# B&R Automation Studio project PLC code - cp (part 17)

#### MachineModel.st
```iecst
ACTION MachineModel:

	//Assignation of machine model just when unnasigned
	IF gMachine.In.iMachineModelCode=0 THEN
		InputsMachineModel;
	END_IF

	// Code To PLC.
	// From the inputs of the type of machine readed by the inputs to the Parameter of the particular Type of Machine
	MachineModelAssignation;

	//Assignation of the axis
	AxisAssignation;

	// Code To Kernel	(Tranfer the other codes)
	MachineModelCodificationToSw;

END_ACTION

ACTION MachineModelAssignation:

	CASE gMachine.Pt.ConfigNameID OF

		GC_CONFIG_2BK12BAR_ID:
			CASE gMachine.In.iMachineModelCode OF
				51: // P4 Large 1 Block		|| 51-> 0011 0011
					gMachine.Pt.MachineModel:= Type_P4_6B_L;				// 3
				15: // P4 Large 2 Block		|| 15-> 0000 1111
					gMachine.Pt.MachineModel:=Type_P4_12B_L;				// 4
				48: // P4 Short 1 Block		|| 48-> 0011 0000
					gMachine.Pt.MachineModel:=Type_P4_6B;					// 1
				11: //S1400 Without Vacuum	|| 11-> 0000 1011
					gMachine.Pt.MachineModel:=Type_P4_CBK;					// 14
				12: // P4 Short 2 Block		|| 12-> 0000 1100
					gMachine.Pt.MachineModel:=Type_P4_12B;					// 2
				52: // P4 Long 1 Block Cubik|| 11-> 0011 0100
					gMachine.Pt.MachineModel:= Type_P4_CBK;				// 12 -->P4 1 Block normal with vacuum and cubik functions
				ELSE
					gMachine.Pt.MachineModel:=NoType;

			END_CASE

		GC_CONFIG_1BK2BAR_ID:
			CASE gMachine.In.iMachineModelCode OF
				3: // EBRO 1 Block			|| 3->  0000 0011
					gMachine.Pt.MachineModel:=Type_SHLD;					// 5
				ELSE
					gMachine.Pt.MachineModel:=NoType;

			END_CASE

		GC_CONFIG_BM_1BK8BAR_ID:
			CASE gMachine.In.iMachineModelCode OF
				5: //P5 Oil					|| 5->	0000 0101
					gMachine.Pt.MachineModel:=Type_P5_OIL;
				6: //P5 Water				|| 6->	0000 0110
					gMachine.Pt.MachineModel:=Type_P5_WTR;
				13: //S1400 Without Vacuum	|| 13-> 0000 1101
					gMachine.Pt.MachineModel:=Type_S1400;
				14: //S1400 With Vacuum	PWRLNK	|| 14->	0000 1110
					gMachine.Pt.MachineModel:=Type_S1400_VAC_PWRLNK;
				15: //S1400 With Vacuum	CAN		|| 14->	0000 1111
					gMachine.Pt.MachineModel:=Type_S1400_VAC_CAN;

				ELSE
					gMachine.Pt.MachineModel:=NoType;

			END_CASE

		GC_CONFIG_1BK8BAR_NOZ2_ID:
			CASE gMachine.In.iMachineModelCode OF
				40:
					gMachine.Pt.MachineModel:=Type_NOZ_2_UV;				// 15
				41:
					gMachine.Pt.MachineModel:=Type_NOZ_2_UV_White;

				ELSE
					gMachine.Pt.MachineModel:=NoType;

			END_CASE

		GC_CONFIG_1BK8BAR_NOZ2_AQ_ID:
			CASE gMachine.In.iMachineModelCode OF
				39:
					gMachine.Pt.MachineModel:=Type_NOZ_2_AQ;

				ELSE
					gMachine.Pt.MachineModel:=NoType;

			END_CASE

		GC_CONFIG_1BK7BAR_CUBE_ID:
			CASE gMachine.In.iMachineModelCode OF
				01:
					gMachine.Pt.MachineModel:=Type_CUBE_INSPECTION;
				02:
					gMachine.Pt.MachineModel := Type_CUBE_GULLIVER_INSPECTION;
				04:
					gMachine.Pt.MachineModel:=Type_CUBE;
				08:
					gMachine.Pt.MachineModel := Type_CUBE_GULLIVER;
				ELSE
					gMachine.Pt.MachineModel:=NoType;

			END_CASE

		GC_CONFIG_1BK10BAR_MECANO_ID:
			CASE gMachine.In.iMachineModelCode OF
				60:
					gMachine.Pt.MachineModel:=Type_MECANO_UV_WHITE;
				61:
					gMachine.Pt.MachineModel:=Type_MECANO_UV_OPV;
				62:
					gMachine.Pt.MachineModel:=Type_MECANO_UV_WHITE_OPV;

				ELSE
					gMachine.Pt.MachineModel:=NoType;

			END_CASE

		GC_CONFIG_SIMTEST_ID:
			CASE gMachine.In.iMachineModelCode OF
				51: // P4 Large 1 Block		|| 51-> 0011 0011
					gMachine.Pt.MachineModel:= Type_P4_6B_L;				// 3
				15: // P4 Large 2 Block		|| 15-> 0000 1111
					gMachine.Pt.MachineModel:=Type_P4_12B_L;				// 4
				48: // P4 Short 1 Block		|| 48-> 0011 0000
					gMachine.Pt.MachineModel:=Type_P4_6B;					// 1
				12: // P4 Short 2 Block		|| 12-> 0000 0011
					gMachine.Pt.MachineModel:=Type_P4_12B;					// 2
				3: // EBRO 1 Block			|| 3->  0000 0011
					gMachine.Pt.MachineModel:=Type_SHLD;					// 5
				13: //S1400 Without Vacuum	|| 13-> 0000 1011
					gMachine.Pt.MachineModel:=Type_S1400;					// 9
				14: //S1400 With Vacuum	PWLNK
					gMachine.Pt.MachineModel:=Type_S1400_VAC_PWRLNK;
				1015: //S1400 With Vacuum CAN
					gMachine.Pt.MachineModel:=Type_S1400_VAC_PWRLNK;
				52: // P4 Long 1 Block Cubik|| 11-> 0011 0100
					gMachine.Pt.MachineModel:= Type_P4_CBK;				// 12 -->P4 1 Block normal with vacuum and cubik functions
				5: //P5 Oil					|| 5->	0000 0101
					gMachine.Pt.MachineModel:=Type_P5_OIL;					// 12
				6: //P5 Water				|| 6->	0000 0110
					gMachine.Pt.MachineModel:=Type_P5_WTR;					// 13
				11: //S1400 Without Vacuum	|| 11-> 0000 1011
					gMachine.Pt.MachineModel:=Type_P4_CBK;					// 14
				39:
					gMachine.Pt.MachineModel:=Type_NOZ_2_AQ;					// 11
				40:
					gMachine.Pt.MachineModel:=Type_NOZ_2_UV;				// 15
				41:
					gMachine.Pt.MachineModel:=Type_NOZ_2_UV_White;
				60:
					gMachine.Pt.MachineModel:=Type_MECANO_UV_WHITE;
				61:
					gMachine.Pt.MachineModel:=Type_MECANO_UV_OPV;
				62:
					gMachine.Pt.MachineModel:=Type_MECANO_UV_WHITE_OPV;

				10001:
					gMachine.Pt.MachineModel := Type_CUBE;
				10002:
					gMachine.Pt.MachineModel := Type_CUBE_GULLIVER;
				10003:
					gMachine.Pt.MachineModel := Type_CUBE_INSPECTION;
				10004:
					gMachine.Pt.MachineModel := Type_CUBE_GULLIVER_INSPECTION;

				ELSE
					gMachine.Pt.MachineModel:=NoType;

			END_CASE
			xChangedSimMachine := simMachine_copy <> gSimMachine.Parameters.MachineType;
			simMachine_copy := gSimMachine.Parameters.MachineType;

		ELSE
			gMachine.Pt.MachineModel:=NoType;

	END_CASE

END_ACTION

ACTION AxisAssignation:

	IF gMachine.Pt.ConfigNameID = GC_CONFIG_SIMTEST_ID THEN
		Axis_Simulation;
		RETURN;
	END_IF

    //Name of the Axis as defined in Hardware
	CASE gMachine.Pt.MachineModel OF

		Type_P4_6B,
		Type_P4_6B_L,
		Type_P4_12B,
		Type_P4_12B_L:
			Axis_P4;

		Type_SHLD,
		Type_SHLD_L:
			Axis_Shield;

		Type_S1400,
		Type_S1400_VAC_PWRLNK,
		Type_S1400_VAC_CAN:
			Axis_S1400;

		Type_P5_OIL,
		Type_P5_WTR:
			Axis_P5;

		Type_NOZ_2_AQ:
			Axis_Nozomi2_AQ;

		Type_NOZ_2_UV,
		Type_NOZ_2_UV_White:
			Axis_Nozomi2;

		Type_CUBE,
		Type_CUBE_INSPECTION,
		Type_CUBE_GULLIVER,
		Type_CUBE_GULLIVER_INSPECTION:
			Axis_Cube;

		Type_MECANO_UV_WHITE,
		Type_MECANO_UV_OPV,
		Type_MECANO_UV_WHITE_OPV:
			Axis_Mecano;

		ELSE
			//No machine assigned
			RETURN;

	END_CASE

END_ACTION

ACTION Axis_Simulation:

	gAxis[1].Parameter.Init.AxisObjectName			:=	'gAxis01';	//Instance_Belt
	gAxis[2].Parameter.Init.AxisObjectName			:=	'gAxis21';	//Instance_BK1
	gAxis[3].Parameter.Init.AxisObjectName			:=	'gAxis121';	//Instance_BK2
	gAxis[4].Parameter.Init.AxisObjectName			:=	'gAxisStp01';	//Instance_Front3L
	gAxis[5].Parameter.Init.AxisObjectName			:=	'gAxisStp02';	//Instance_Back3L
	gAxis[6].Parameter.Init.AxisObjectName			:=	'gAxis41';	//Instance_NonCrash1

	// Assignation of Master axis
	gAxis[5].Parameter.Init.MasterGearObjectName	:=	'gAxisStp01';	//Instance_Front3L

	LoadDefaultServoConfig(ADR(gAxis[1]));
	LoadDefaultServoConfig(ADR(gAxis[2]));
	LoadDefaultServoConfig(ADR(gAxis[3]));
	LoadDefaultStepperConfig(ADR(gAxis[4])); //These are steppers and do not have torque
	LoadDefaultStepperConfig(ADR(gAxis[5])); //These are steppers and do not have torque
	LoadDefaultServoConfig(ADR(gAxis[6]));

	//Assign comms type of inverters depending on the machine type
	CASE gMachine.Pt.MachineModel OF
		Type_S1400_VAC_PWRLNK:
			gAxisInverter[1].Parameters.CommsType := COMMS_POWERLINK;
			gAxisInverter[2].Parameters.CommsType := COMMS_POWERLINK;
			gAxisInverter[3].Parameters.CommsType := COMMS_POWERLINK;
			gAxisInverter[4].Parameters.CommsType := COMMS_POWERLINK;

		Type_NOZ_2_AQ:
			IF X20IF1072_SS3.ModuleOk THEN
				gAxisInverter[1].Parameters.CommsType := COMMS_CANOPEN;
				gAxisInverter[2].Parameters.CommsType := COMMS_CANOPEN;
				gAxisInverter[3].Parameters.CommsType := COMMS_CANOPEN;
				gAxisInverter[4].Parameters.CommsType := COMMS_CANOPEN;
			ELSE
				gAxisInverter[1].Parameters.CommsType := COMMS_POWERLINK;
				gAxisInverter[2].Parameters.CommsType := COMMS_POWERLINK;
				gAxisInverter[3].Parameters.CommsType := COMMS_POWERLINK;
				gAxisInverter[4].Parameters.CommsType := COMMS_POWERLINK;
			END_IF

		Type_NOZ_2_UV,
		Type_NOZ_2_UV_White:
			IF X20IF1072_SS1.ModuleOk THEN
				gAxisInverter[1].Parameters.CommsType := COMMS_CANOPEN;
				gAxisInverter[2].Parameters.CommsType := COMMS_CANOPEN;
				gAxisInverter[3].Parameters.CommsType := COMMS_CANOPEN;
				gAxisInverter[4].Parameters.CommsType := COMMS_CANOPEN;
			ELSE
				gAxisInverter[1].Parameters.CommsType := COMMS_POWERLINK;
				gAxisInverter[2].Parameters.CommsType := COMMS_POWERLINK;
				gAxisInverter[3].Parameters.CommsType := COMMS_POWERLINK;
				gAxisInverter[4].Parameters.CommsType := COMMS_POWERLINK;
			END_IF

		Type_CUBE,
		Type_CUBE_INSPECTION,
		Type_CUBE_GULLIVER,
		Type_CUBE_GULLIVER_INSPECTION:
			gAxisInverter[1].Parameters.CommsType := COMMS_POWERLINK;
			gAxisInverter[2].Parameters.CommsType := COMMS_POWERLINK;
			gAxisInverter[3].Parameters.CommsType := COMMS_POWERLINK;

		Type_MECANO_UV_WHITE,
		Type_MECANO_UV_OPV,
		Type_MECANO_UV_WHITE_OPV:
			gAxisInverter[1].Parameters.CommsType := COMMS_POWERLINK;
			gAxisInverter[2].Parameters.CommsType := COMMS_POWERLINK;
			gAxisInverter[3].Parameters.CommsType := COMMS_POWERLINK;
			gAxisInverter[4].Parameters.CommsType := COMMS_POWERLINK;

	END_CASE
	gAxisInverter[1].Parameters.Hardware.CpuFamily := gMachine.St.HwData.Family;
	gAxisInverter[2].Parameters.Hardware.CpuFamily := gMachine.St.HwData.Family;
	gAxisInverter[3].Parameters.Hardware.CpuFamily := gMachine.St.HwData.Family;
	gAxisInverter[4].Parameters.Hardware.CpuFamily := gMachine.St.HwData.Family;

	//This is the physical node of each Icla
	gIcla[1].Parameter.Node:=5;
	gIcla[1].Parameter.Network := 'IF7';
	gIcla[2].Parameter.Node:=7;
	gIcla[2].Parameter.Network := 'IF7';
	gIcla[3].Parameter.Node:=50; //Same node number than in Nozomi C18000
	gIcla[3].Parameter.Network := 'IF7';

END_ACTION

ACTION Axis_P4:

	gAxis[1].Parameter.Init.AxisObjectName			:=	'gAxis01';	//Instance_Belt
	gAxis[2].Parameter.Init.AxisObjectName			:=	'gAxis21';	//Instance_BK1
	gAxis[3].Parameter.Init.AxisObjectName			:=	'gAxis121';	//Instance_BK2
	gAxis[4].Parameter.Init.AxisObjectName			:=	'gAxisStp01';	//Instance_Front3L
	gAxis[5].Parameter.Init.AxisObjectName			:=	'gAxisStp02';	//Instance_Back3L

	// Assignation of Master axis
	gAxis[5].Parameter.Init.MasterGearObjectName	:=	'gAxisStp01';	//Instance_Front3L

	LoadDefaultServoConfig(ADR(gAxis[1]));
	LoadDefaultServoConfig(ADR(gAxis[2]));
	LoadDefaultServoConfig(ADR(gAxis[3]));
	LoadDefaultStepperConfig(ADR(gAxis[4])); //These are steppers and do not have torque
	LoadDefaultStepperConfig(ADR(gAxis[5])); //These are steppers and do not have torque

	//This is the physical node of each Icla
	gIcla[1].Parameter.Node:=5;
	gIcla[1].Parameter.Network := 'IF7';
	gIcla[1].Parameter.xAutoresetComms := TRUE;
	gIcla[2].Parameter.Node:=7;
	gIcla[2].Parameter.Network := 'IF7';
	gIcla[2].Parameter.xAutoresetComms := TRUE;

END_ACTION

ACTION Axis_Shield:

	gAxis[1].Parameter.Init.AxisObjectName			:=	'gAxis01';	//Instance_Belt
	gAxis[2].Parameter.Init.AxisObjectName			:=	'gAxis21';	//Instance_BK1
	gAxis[3].Parameter.Init.AxisObjectName			:=	'gAxisStp01';	//Instance_Front3L
	gAxis[4].Parameter.Init.AxisObjectName			:=	'gAxisStp02';	//Instance_Back3L

	// Assignation of Master axis
	gAxis[4].Parameter.Init.MasterGearObjectName	:=	'gAxisStp01';	//Instance_Front3L

	LoadDefaultServoConfig(ADR(gAxis[1]));
	LoadDefaultServoConfig(ADR(gAxis[2]));
	LoadDefaultStepperConfig(ADR(gAxis[3])); //These are steppers and do not have torque
	LoadDefaultStepperConfig(ADR(gAxis[4])); //These are steppers and do not have torque

	//This is the physical node of each Icla
	gIcla[1].Parameter.Node:=5;
	gIcla[1].Parameter.Network := 'IF7';
	gIcla[1].Parameter.xAutoresetComms := TRUE;

END_ACTION

ACTION Axis_S1400:

	gAxis[1].Parameter.Init.AxisObjectName			:=	'gAxis01';	//Instance_Belt
	gAxis[2].Parameter.Init.AxisObjectName			:=	'gAxis21';	//Instance_BK1
	gAxis[3].Parameter.Init.AxisObjectName			:=	'gAxisStp01';	//Instance_Front3L
	gAxis[4].Parameter.Init.AxisObjectName			:=	'gAxisStp02';	//Instance_Back3L
	gAxis[5].Parameter.Init.AxisObjectName			:=	'gAxis41';	//Instance_NonCrash1

	// Assignation of Master axis
	gAxis[4].Parameter.Init.MasterGearObjectName	:=	'gAxisStp01';	//Instance_Front3L

	CASE gMachine.Pt.MachineModel OF
		Type_S1400_VAC_PWRLNK:
			gAxisInverter[1].Parameters.Hardware.PowerLinkInterface := 'IF3';
			gAxisInverter[1].Parameters.Hardware.Node := 81;
			gAxisInverter[1].Parameters.AccelerationTime := 1;
			gAxisInverter[1].Parameters.DecelerationTime := 1;
			gAxisInverter[1].Parameters.CommsType := COMMS_POWERLINK;
			gAxisInverter[2].Parameters.Hardware.PowerLinkInterface := 'IF3';
			gAxisInverter[2].Parameters.Hardware.Node := 82;
			gAxisInverter[2].Parameters.AccelerationTime := 1;
			gAxisInverter[2].Parameters.DecelerationTime := 1;
			gAxisInverter[2].Parameters.CommsType := COMMS_POWERLINK;
			gAxisInverter[3].Parameters.Hardware.PowerLinkInterface := 'IF3';
			gAxisInverter[3].Parameters.Hardware.Node := 83;
			gAxisInverter[3].Parameters.AccelerationTime := 1;
			gAxisInverter[3].Parameters.DecelerationTime := 1;
			gAxisInverter[3].Parameters.CommsType := COMMS_POWERLINK;
			gAxisInverter[4].Parameters.Hardware.PowerLinkInterface := 'IF3';
			gAxisInverter[4].Parameters.Hardware.Node := 84;
			gAxisInverter[4].Parameters.AccelerationTime := 1;
			gAxisInverter[4].Parameters.DecelerationTime := 1;
			gAxisInverter[4].Parameters.CommsType := COMMS_POWERLINK;

		Type_S1400_VAC_CAN:
			gAxisInverter[1].Parameters.CommsType := COMMS_CANOPEN;
			gAxisInverter[2].Parameters.CommsType := COMMS_CANOPEN;
			gAxisInverter[3].Parameters.CommsType := COMMS_CANOPEN;
			gAxisInverter[4].Parameters.CommsType := COMMS_CANOPEN;

	END_CASE

	gAxisInverter[1].Parameters.Hardware.CpuFamily := gMachine.St.HwData.Family;
	gAxisInverter[2].Parameters.Hardware.CpuFamily := gMachine.St.HwData.Family;
	gAxisInverter[3].Parameters.Hardware.CpuFamily := gMachine.St.HwData.Family;
	gAxisInverter[4].Parameters.Hardware.CpuFamily := gMachine.St.HwData.Family;

	LoadDefaultServoConfig(ADR(gAxis[1]));
	LoadDefaultServoConfig(ADR(gAxis[2]));
	LoadDefaultStepperConfig(ADR(gAxis[3])); //These are steppers and do not have torque
	LoadDefaultStepperConfig(ADR(gAxis[4])); //These are steppers and do not have torque
	LoadDefaultServoConfig(ADR(gAxis[5]));

	//This is the physical node of each Icla
	gIcla[1].Parameter.Node:=5;
	gIcla[1].Parameter.Network := 'IF7';
	gIcla[1].Parameter.xAutoresetComms := TRUE;

END_ACTION

ACTION Axis_P5:

	gAxis[1].Parameter.Init.AxisObjectName			:=	'gAxis02';	//Instance_Belt
	gAxis[2].Parameter.Init.AxisObjectName			:=	'gAxis21';	//Instance_BK1
	gAxis[3].Parameter.Init.AxisObjectName			:=	'gAxisStp01';	//Instance_Front3L
	gAxis[4].Parameter.Init.AxisObjectName			:=	'gAxisStp02';	//Instance_Back3L

	// Assignation of Master axis
	gAxis[4].Parameter.Init.MasterGearObjectName	:=	'gAxisStp01';	//Instance_Front3L

	LoadDefaultServoConfig(ADR(gAxis[1]));
	LoadDefaultServoConfig(ADR(gAxis[2]));
	LoadDefaultStepperConfig(ADR(gAxis[3])); //These are steppers and do not have torque
	LoadDefaultStepperConfig(ADR(gAxis[4])); //These are steppers and do not have torque

	//This is the physical node of each Icla
	gIcla[1].Parameter.Node:=5;
	gIcla[1].Parameter.Network := 'IF7';
	gIcla[1].Parameter.xAutoresetComms := TRUE;

END_ACTION

ACTION Axis_Nozomi2:

	gAxis[1].Parameter.Init.AxisObjectName			:=	'gAxis01';	//Instance_Belt
	gAxis[2].Parameter.Init.AxisObjectName			:=	'gAxis21';	//Instance_BK1

	LoadDefaultServoConfig(ADR(gAxis[1]));
	LoadDefaultServoConfig(ADR(gAxis[2]));

	CASE gMachine.Pt.MachineModel OF
		Type_NOZ_2_UV,
		Type_NOZ_2_UV_White:

			IF X20IF1072_SS1.ModuleOk THEN
				gAxisInverter[1].Parameters.CommsType := COMMS_CANOPEN;
				gAxisInverter[1].Parameters.Hardware.Node := 81;
				gAxisInverter[1].Parameters.Hardware.PowerLinkInterface := 'IF1';
				gAxisInverter[2].Parameters.CommsType := COMMS_CANOPEN;
				gAxisInverter[2].Parameters.Hardware.Node := 82;
				gAxisInverter[2].Parameters.Hardware.PowerLinkInterface := 'IF1';
				gAxisInverter[3].Parameters.CommsType := COMMS_CANOPEN;
				gAxisInverter[3].Parameters.Hardware.Node := 83;
				gAxisInverter[3].Parameters.Hardware.PowerLinkInterface := 'IF1';
				gAxisInverter[4].Parameters.CommsType := COMMS_CANOPEN;
				gAxisInverter[4].Parameters.Hardware.Node := 84;
				gAxisInverter[4].Parameters.Hardware.PowerLinkInterface := 'IF1';
			ELSE
				gAxisInverter[1].Parameters.Hardware.PowerLinkInterface := 'IF3';
				gAxisInverter[1].Parameters.Hardware.Node := 81;
				gAxisInverter[1].Parameters.AccelerationTime := 3;
				gAxisInverter[1].Parameters.DecelerationTime := 1;
				gAxisInverter[1].Parameters.CommsType := COMMS_POWERLINK;
				gAxisInverter[2].Parameters.Hardware.PowerLinkInterface := 'IF3';
				gAxisInverter[2].Parameters.Hardware.Node := 82;
				gAxisInverter[2].Parameters.AccelerationTime := gAxisInverter[1].Parameters.AccelerationTime;
				gAxisInverter[2].Parameters.DecelerationTime := gAxisInverter[1].Parameters.DecelerationTime;
				gAxisInverter[2].Parameters.CommsType := COMMS_POWERLINK;
				gAxisInverter[3].Parameters.Hardware.PowerLinkInterface := 'IF3';
				gAxisInverter[3].Parameters.Hardware.Node := 83;
				gAxisInverter[3].Parameters.AccelerationTime := gAxisInverter[1].Parameters.AccelerationTime;
				gAxisInverter[3].Parameters.DecelerationTime := gAxisInverter[1].Parameters.DecelerationTime;
				gAxisInverter[3].Parameters.CommsType := COMMS_POWERLINK;
				gAxisInverter[4].Parameters.Hardware.PowerLinkInterface := 'IF3';
				gAxisInverter[4].Parameters.Hardware.Node := 84;
				gAxisInverter[4].Parameters.AccelerationTime := gAxisInverter[1].Parameters.AccelerationTime;
				gAxisInverter[4].Parameters.DecelerationTime := gAxisInverter[1].Parameters.DecelerationTime;
				gAxisInverter[4].Parameters.CommsType := COMMS_POWERLINK;
			END_IF

	END_CASE

	gAxisInverter[1].Parameters.Hardware.CpuFamily := gMachine.St.HwData.Family;
	gAxisInverter[2].Parameters.Hardware.CpuFamily := gMachine.St.HwData.Family;
	gAxisInverter[3].Parameters.Hardware.CpuFamily := gMachine.St.HwData.Family;
	gAxisInverter[4].Parameters.Hardware.CpuFamily := gMachine.St.HwData.Family;

	//This is the physical node of each Icla
	gIcla[1].Parameter.Node:=5;
	gIcla[1].Parameter.Network := 'IF7';
	gIcla[1].Parameter.xAutoresetComms := TRUE;
	gIcla[2].Parameter.Node:=2; //50; [RGP] We had to change number node to match the node order that AS was expecting. Escalated to JNovella. No reason explained.
	gIcla[2].Parameter.Network := 'IF7';
	gIcla[2].Parameter.xAutoresetComms := TRUE;
	gIcla[3].Parameter.Node:=6;
	gIcla[3].Parameter.Network := 'IF7';
	gIcla[3].Parameter.xAutoresetComms := TRUE;
	gIcla[4].Parameter.Node:=7;
	gIcla[4].Parameter.Network := 'IF7';
	gIcla[4].Parameter.xAutoresetComms := TRUE;
	gIcla[5].Parameter.Node:=8;
	gIcla[5].Parameter.Network := 'IF7';
	gIcla[5].Parameter.xAutoresetComms := TRUE;
	gIcla[6].Parameter.Node:=9;
	gIcla[6].Parameter.Network := 'IF7';
	gIcla[6].Parameter.xAutoresetComms := TRUE;

END_ACTION

ACTION Axis_Nozomi2_AQ:

	gAxis[1].Parameter.Init.AxisObjectName			:=	'gAxis01';	//Instance_Belt
	gAxis[2].Parameter.Init.AxisObjectName			:=	'gAxis21';	//Instance_BK1

	LoadDefaultServoConfig(ADR(gAxis[1]));
	LoadDefaultServoConfig(ADR(gAxis[2]));

	CASE gMachine.Pt.MachineModel OF
		Type_NOZ_2_AQ:

			IF X20IF1072_SS3.ModuleOk THEN
				gAxisInverter[1].Parameters.CommsType := COMMS_CANOPEN;
				gAxisInverter[1].Parameters.Hardware.Node := 81;
				gAxisInverter[1].Parameters.Hardware.PowerLinkInterface := 'SS3.IF1';
				gAxisInverter[2].Parameters.CommsType := COMMS_CANOPEN;
				gAxisInverter[2].Parameters.Hardware.Node := 82;
				gAxisInverter[2].Parameters.Hardware.PowerLinkInterface := 'SS3.IF1';
				gAxisInverter[3].Parameters.CommsType := COMMS_CANOPEN;
				gAxisInverter[3].Parameters.Hardware.Node := 83;
				gAxisInverter[3].Parameters.Hardware.PowerLinkInterface := 'SS3.IF1';
				gAxisInverter[4].Parameters.CommsType := COMMS_CANOPEN;
				gAxisInverter[4].Parameters.Hardware.Node := 84;
				gAxisInverter[4].Parameters.Hardware.PowerLinkInterface := 'SS3.IF1';
			ELSE
				gAxisInverter[1].Parameters.Hardware.PowerLinkInterface := 'IF3';
				gAxisInverter[1].Parameters.Hardware.Node := 81;
				gAxisInverter[1].Parameters.AccelerationTime := 3;
				gAxisInverter[1].Parameters.DecelerationTime := 1;
				gAxisInverter[1].Parameters.CommsType := COMMS_POWERLINK;
				gAxisInverter[2].Parameters.Hardware.PowerLinkInterface := 'IF3';
				gAxisInverter[2].Parameters.Hardware.Node := 82;
				gAxisInverter[2].Parameters.AccelerationTime := gAxisInverter[1].Parameters.AccelerationTime;
				gAxisInverter[2].Parameters.DecelerationTime := gAxisInverter[1].Parameters.DecelerationTime;
				gAxisInverter[2].Parameters.CommsType := COMMS_POWERLINK;
				gAxisInverter[3].Parameters.Hardware.PowerLinkInterface := 'IF3';
				gAxisInverter[3].Parameters.Hardware.Node := 83;
				gAxisInverter[3].Parameters.AccelerationTime := gAxisInverter[1].Parameters.AccelerationTime;
				gAxisInverter[3].Parameters.DecelerationTime := gAxisInverter[1].Parameters.DecelerationTime;
				gAxisInverter[3].Parameters.CommsType := COMMS_POWERLINK;
				gAxisInverter[4].Parameters.Hardware.PowerLinkInterface := 'IF3';
				gAxisInverter[4].Parameters.Hardware.Node := 84;
				gAxisInverter[4].Parameters.AccelerationTime := gAxisInverter[1].Parameters.AccelerationTime;
				gAxisInverter[4].Parameters.DecelerationTime := gAxisInverter[1].Parameters.DecelerationTime;
				gAxisInverter[4].Parameters.CommsType := COMMS_POWERLINK;
			END_IF

	END_CASE

	gAxisInverter[1].Parameters.Hardware.CpuFamily := gMachine.St.HwData.Family;
	gAxisInverter[2].Parameters.Hardware.CpuFamily := gMachine.St.HwData.Family;
	gAxisInverter[3].Parameters.Hardware.CpuFamily := gMachine.St.HwData.Family;
	gAxisInverter[4].Parameters.Hardware.CpuFamily := gMachine.St.HwData.Family;

	//This is the physical node of each Icla
	gIcla[1].Parameter.Node:=5;
	gIcla[1].Parameter.Network := 'SS2.IF1';
	gIcla[1].Parameter.xAutoresetComms := TRUE;
	gIcla[2].Parameter.Node:=2; //50; [RGP] We had to change number node to match the node order that AS was expecting. Escalated to JNovella. No reason explained.
	gIcla[2].Parameter.Network := 'SS2.IF1';
	gIcla[2].Parameter.xAutoresetComms := TRUE;
	gIcla[3].Parameter.Node:=6;
	gIcla[3].Parameter.Network := 'SS2.IF1';
	gIcla[3].Parameter.xAutoresetComms := TRUE;
	gIcla[4].Parameter.Node:=7;
	gIcla[4].Parameter.Network := 'SS2.IF1';
	gIcla[4].Parameter.xAutoresetComms := TRUE;
	gIcla[5].Parameter.Node:=8;
	gIcla[5].Parameter.Network := 'SS2.IF1';
	gIcla[5].Parameter.xAutoresetComms := TRUE;
	gIcla[6].Parameter.Node:=9;
	gIcla[6].Parameter.Network := 'SS2.IF1';
	gIcla[6].Parameter.xAutoresetComms := TRUE;

END_ACTION

ACTION Axis_Cube:

	gAxis[1].Parameter.Init.AxisObjectName			:=	'gAxis01';	//Instance_Belt
	gAxis[2].Parameter.Init.AxisObjectName			:=	'gAxis21';	//Instance_BK1

	LoadDefaultServoConfig(ADR(gAxis[1]));
	LoadDefaultServoConfig(ADR(gAxis[2]));

	CASE gMachine.Pt.MachineModel OF
		Type_CUBE,
		Type_CUBE_INSPECTION,
		Type_CUBE_GULLIVER,
		Type_CUBE_GULLIVER_INSPECTION:

			gAxisInverter[1].Parameters.Hardware.PowerLinkInterface := 'IF3';
			gAxisInverter[1].Parameters.Hardware.Node := 81;
			gAxisInverter[1].Parameters.AccelerationTime := 0;
			gAxisInverter[1].Parameters.DecelerationTime := 0;
			gAxisInverter[1].Parameters.CommsType := COMMS_POWERLINK;
			gAxisInverter[1].Parameters.Type := INV_ABB;
			gAxisInverter[1].Parameters.ControlMode := 0;
			gAxisInverter[2].Parameters.Hardware.PowerLinkInterface := 'IF3';
			gAxisInverter[2].Parameters.Hardware.Node := 82;
			gAxisInverter[2].Parameters.AccelerationTime := 0;
			gAxisInverter[2].Parameters.DecelerationTime := 0;
			gAxisInverter[2].Parameters.CommsType := COMMS_POWERLINK;
			gAxisInverter[2].Parameters.Type := INV_ABB;
			gAxisInverter[2].Parameters.ControlMode := 0;

			gAxisInverter[3].Parameters.Hardware.PowerLinkInterface := 'IF3';
			gAxisInverter[3].Parameters.Hardware.Node := 91;
			gAxisInverter[3].Parameters.AccelerationTime := 0;
			gAxisInverter[3].Parameters.DecelerationTime := 0;
			gAxisInverter[3].Parameters.CommsType := COMMS_POWERLINK;
			gAxisInverter[3].Parameters.Type := INV_ABB;
			gAxisInverter[3].Parameters.ControlMode := 0;

	END_CASE

	gAxisInverter[1].Parameters.Hardware.CpuFamily := gMachine.St.HwData.Family;
	gAxisInverter[2].Parameters.Hardware.CpuFamily := gMachine.St.HwData.Family;
	gAxisInverter[3].Parameters.Hardware.CpuFamily := gMachine.St.HwData.Family;

	//This is the physical node of each Icla
	gIcla[1].Parameter.Node:=5;
	gIcla[1].Parameter.Network := 'SS2.IF1';
	gIcla[1].Parameter.xAutoresetComms := TRUE;

END_ACTION

ACTION Axis_Mecano:

	gAxis[1].Parameter.Init.AxisObjectName			:=	'gAxis01';	//Instance_Belt
	gAxis[2].Parameter.Init.AxisObjectName			:=	'gAxis21';	//Instance_BK1

	LoadDefaultServoConfig(ADR(gAxis[1]));
	LoadDefaultServoConfig(ADR(gAxis[2]));

	gAxisInverter[1].Parameters.Hardware.PowerLinkInterface := 'IF3';
	gAxisInverter[1].Parameters.Hardware.Node := 81;
	gAxisInverter[1].Parameters.AccelerationTime := 0;
	gAxisInverter[1].Parameters.DecelerationTime := 0;
	gAxisInverter[1].Parameters.CommsType := COMMS_POWERLINK;
	gAxisInverter[1].Parameters.Type := INV_ABB;
	gAxisInverter[1].Parameters.ControlMode := 0;
	gAxisInverter[2].Parameters.Hardware.PowerLinkInterface := 'IF3';
	gAxisInverter[2].Parameters.Hardware.Node := 82;
	gAxisInverter[2].Parameters.AccelerationTime := 0;
	gAxisInverter[2].Parameters.DecelerationTime := 0;
	gAxisInverter[2].Parameters.CommsType := COMMS_POWERLINK;
	gAxisInverter[2].Parameters.Type := INV_ABB;
	gAxisInverter[2].Parameters.ControlMode := 0;
	gAxisInverter[3].Parameters.Hardware.PowerLinkInterface := 'IF3';
	gAxisInverter[3].Parameters.Hardware.Node := 83;
	gAxisInverter[3].Parameters.AccelerationTime := 0;
	gAxisInverter[3].Parameters.DecelerationTime := 0;
	gAxisInverter[3].Parameters.CommsType := COMMS_POWERLINK;
	gAxisInverter[3].Parameters.Type := INV_ABB;
	gAxisInverter[3].Parameters.ControlMode := 0;
	gAxisInverter[4].Parameters.Hardware.PowerLinkInterface := 'IF3';
	gAxisInverter[4].Parameters.Hardware.Node := 84;
	gAxisInverter[4].Parameters.AccelerationTime := 0;
	gAxisInverter[4].Parameters.DecelerationTime := 0;
	gAxisInverter[4].Parameters.CommsType := COMMS_POWERLINK;
	gAxisInverter[4].Parameters.Type := INV_ABB;
	gAxisInverter[4].Parameters.ControlMode := 0;

	gAxisInverter[1].Parameters.Hardware.CpuFamily := gMachine.St.HwData.Family;
	gAxisInverter[2].Parameters.Hardware.CpuFamily := gMachine.St.HwData.Family;
	gAxisInverter[3].Parameters.Hardware.CpuFamily := gMachine.St.HwData.Family;
	gAxisInverter[4].Parameters.Hardware.CpuFamily := gMachine.St.HwData.Family;

	//This is the physical node of each Icla
	gIcla[1].Parameter.Node:=5;
	gIcla[1].Parameter.Network := 'SS2.IF1';
	gIcla[1].Parameter.xAutoresetComms := TRUE;
	gIcla[2].Parameter.Node:=2; //50; [RGP] We had to change number node to match the node order that AS was expecting. Escalated to JNovella. No reason explained.
	gIcla[2].Parameter.Network := 'SS2.IF1';
	gIcla[2].Parameter.xAutoresetComms := TRUE;
	gIcla[3].Parameter.Node:=6;
	gIcla[3].Parameter.Network := 'SS2.IF1';
	gIcla[3].Parameter.xAutoresetComms := TRUE;
	gIcla[4].Parameter.Node:=7;
	gIcla[4].Parameter.Network := 'SS2.IF1';
	gIcla[4].Parameter.xAutoresetComms := TRUE;
	gIcla[5].Parameter.Node:=8;
	gIcla[5].Parameter.Network := 'SS2.IF1';
	gIcla[5].Parameter.xAutoresetComms := TRUE;
	gIcla[6].Parameter.Node:=9;
	gIcla[6].Parameter.Network := 'SS2.IF1';
	gIcla[6].Parameter.xAutoresetComms := TRUE;

END_ACTION

ACTION MachineModelCodificationToSw:

	CASE gMachine.Pt.MachineModel OF
		Type_P4_12B:
			gMachine.St.iMachineModelCodeSW:=120;

		Type_P4_12B_L:
			gMachine.St.iMachineModelCodeSW:=150;

		Type_P4_6B:
			gMachine.St.iMachineModelCodeSW:=480;

		Type_P4_CBK,
		Type_P4_6B_L:
			gMachine.St.iMachineModelCodeSW:=510;

		Type_SHLD:
			gMachine.St.iMachineModelCodeSW:=3;

		Type_SHLD_L:
			gMachine.St.iMachineModelCodeSW:=5;

		Type_NOZ_2_AQ:
			gMachine.St.iMachineModelCodeSW:=39;

		Type_NOZ_2_UV,
		Type_NOZ_2_UV_White:
			gMachine.St.iMachineModelCodeSW:=40;

		Type_S1400,
		Type_S1400_VAC_PWRLNK,
		Type_S1400_VAC_CAN,
		Type_P5_OIL,
		Type_P5_WTR:
			gMachine.St.iMachineModelCodeSW:=14;

		Type_CUBE:
			gMachine.St.iMachineModelCodeSW:=1101;

		Type_CUBE_GULLIVER:
			gMachine.St.iMachineModelCodeSW:=1102;
		Type_CUBE_INSPECTION:
			gMachine.St.iMachineModelCodeSW:=1103;

		Type_CUBE_GULLIVER_INSPECTION:
			gMachine.St.iMachineModelCodeSW:=1104;

		Type_MECANO_UV_WHITE,
		Type_MECANO_UV_OPV,
		Type_MECANO_UV_WHITE_OPV:
			gMachine.St.iMachineModelCodeSW:=60;

		ELSE
			gMachine.St.iMachineModelCodeSW:= 0;

	END_CASE

END_ACTION
```

### Program Logical/Printer/Config/SavePermanent (IEC)

#### SavePermanent.st - Init, cyclic, exit code
```iecst
PROGRAM _CYCLIC

	// Permanents Vars
	IF brsstrlen(ADR(gMachine.St.HwData.SerialNumber)) > 0 THEN
		gPermanentSN := gMachine.St.HwData.SerialNumber;
	END_IF
	gPermanentMachine:=gMachine.parSw;
	gPermanentSwBelt:= gBelt.parSw;
	gPermanentBlock[1]:=gBlock[1].parSw;
	gPermanentBlock[2]:=gBlock[2].parSw;
	gPermanentTrVacuum[1] := gTransVacuum[1].parSw;
	gPermanentTrVacuum[2] := gTransVacuum[2].parSw;
	gPermanentAnalogSensor := gDing.State.Permanent;

	FOR iInksIndex:=1 TO MAX_LAST_INK DO
		gPermanentInksParSw[iInksIndex] := gInks[iInksIndex].parSw;
	END_FOR

	gPermanentSimMachinePar:=gSimMachine.Parameters;

	gPermanentVersion.iVersion0 := gPLC.iVersion0;
	gPermanentVersion.iVersion1 := gPLC.iVersion1;
	gPermanentVersion.iVersion2 := gPLC.iVersion2;
	gPermanentVersion.iVersion3 := gPLC.iVersion3;

END_PROGRAM
```

### Package Logical/Printer/MachineCtrl - Controller commads to printer

### Program Logical/Printer/MachineCtrl/MachineCtrl_Fast (IEC)

#### MachineCtrl_Fast.st - Calling program actions
```iecst
PROGRAM _CYCLIC

	//Calculations required previous to execute any action
	Precalculations;

	//Inputs to the machine
	MachineInputs;

	// ACTIONS
	MachineStates;

	// Update status and send more commands
	OrdersPrinter;

	// Reset general alarms
	IF gMachine.AutoCmd.xReset THEN

		//Enable resetting the alarm
		IF gMachine.Al.Alarm.xPDBrokenSensorL1 THEN
			gMachine.Lg.udiPiecesCounterErrorL1 := 0;
		END_IF
		IF gMachine.Al.Alarm.xPDBrokenSensorL2 THEN
			gMachine.Lg.udiPiecesCounterErrorL2 := 0;
		END_IF

		ResetAlarms;
	END_IF

	Alarms;
	AlarmsSummary;

	//Reset Edge commands received from Sw
	gMachine.commandsSw := InputsSwReseted;

	gMachine.St.exec.fast := gMachine.St.exec.fast +1;

END_PROGRAM
```

#### Precalculations.st - Operation/Mode active
```iecst
ACTION Precalculations:

	//To acknowledge whether media thickess has changed
	xMediaThicknessModified := 	rPrevMediaThickness <> gMachine.parSw.Media.rThickness;

	tonEnterSafety.IN := gMachine.In.xSafetyEnabled;
	tonEnterSafety.PT := T#1000ms;
	tonEnterSafety();
	xEdgeSafety := EDGEPOS(tonEnterSafety.Q);

	xBeltMovingPreviousToStop := gBelt.commands.xRunBelt;

END_ACTION
```

#### MachineStates.st - Operation/Mode active
```iecst
ACTION MachineStates:

	// Mute	conditions
	// Impovement in Test:"xRestartAfterPCPLCError": This condition is necessary to remove souns when comnns are restablished

	iReasonAutoCmdStart.0 := gMachine.commandsSw.xStart_GI;
	iReasonAutoCmdStart.1 := tonStartButton.Q AND NOT gMachine.Pt.xDisableStartHoldingGreenButton;

	gMachine.AutoCmd.xStart := EDGEPOS( iReasonAutoCmdStart > 0);

	IF EDGEPOS(gMachine.AutoCmd.xStart) THEN
		LogAutoStart;
	END_IF

	iReasonAutoCmdStop.0 := gMachine.In.Buttons.xStop;
	iReasonAutoCmdStop.1 := gMachine.commandsSw.xStop_GI;
	iReasonAutoCmdStop.2 := gMachine.commandsSw.xToStop_GI;

	IF (NOT gMachine.Pt.xControlledByLine) OR (gLine.Status = LINE_STOPPED) THEN
		gMachine.AutoCmd.xStop  := EDGEPOS(iReasonAutoCmdStop>0);
	ELSE
		gMachine.AutoCmd.xStop  := gMachine.commands.xStop; //Command sent by Line
	END_IF

	IF EDGEPOS(gMachine.AutoCmd.xStop) THEN
		LogAutoStop;
	END_IF

	tofResetAfterEnableSafety(IN:=EDGEPOS(gSafetyController.Outputs.xEnablePrinter1) AND gMachine.Pt.xControlledRemotely, PT:=T#500ms);
	tofToAutoAfterEnableSafety(IN:=EDGEPOS(gMachine.In.xSafetyEnabled), PT:=T#1000ms);
	tofResetFromUI(IN:=gMachine.commandsSw.xReset_GI, PT:=T#100ms);

	gMachine.AutoCmd.xReset:= gMachine.In.Buttons.xReset OR tofResetAfterEnableSafety.Q OR gMachine.commandsSw.xReset_GI;

	gMachine.AutoCmd.xMuteAlarms:= 	gMachine.commandsSw.xMute_GI OR gMachine.In.Buttons.xMute OR gMachine.AutoCmd.xReset;

	IF EDGEPOS(gMachine.commandsSw.xCleanBelt) THEN
		gMachine.AutoCmd.xCleanBelt := TRUE;
	ELSIF gMachine.St.CleaningBelt.xCleaningProcessOnGoing OR (gMachine.St.CleaningBelt.enState = CLN_BELT_ERROR) THEN
		gMachine.AutoCmd.xCleanBelt := FALSE;
	END_IF

	(* Manual/Auto/Zero *)

	// Automatic Mode
	IF  gMachine.In.Buttons.xAuto AND gMachine.St.StartUp.xReadyToAuto AND
		(gMachine.In.Buttons.xReset OR (gMachine.Pt.xControlledRemotely AND (EDGENEG(tofResetFromUI.Q) OR EDGENEG(tofToAutoAfterEnableSafety.Q)))) AND
		NOT gMachine.AlSummary.xAlarmCritical THEN
		        enPrinterState:=PRINTERGEN_AUTO;
	END_IF

	IF enPrinterState = PRINTERGEN_STARTUP AND EDGEPOS(gMachine.St.StartUp.xReadyToAuto) AND
		NOT gMachine.AlSummary.xAlarmCritical THEN
				enPrinterState:=PRINTERGEN_AUTO;
	END_IF

	// StartUp Mode
	IF  gMachine.In.Buttons.xAuto AND gMachine.St.StartUp.Status = STRUP_NOT_STARTED AND
		EDGENEG(tofToAutoAfterEnableSafety.Q) THEN
				enPrinterState:=PRINTERGEN_STARTUP;
	END_IF

	// Manual Mode
	IF	gMachine.In.Buttons.xManual AND gMachine.In.Buttons.xReset THEN
		enPrinterState:=PRINTERGEN_MANUAL;
	END_IF

	// Zero Mode
	iReasonOut.0 := gMachine.In.Buttons.xZero;
	iReasonOut.1 := NOT gMachine.In.Buttons.xAuto AND NOT gMachine.In.Buttons.xManual; // It avoids manual state when safety is NOT ready
	iReasonOut.2 := gMachine.AlSummary.xAlarmCritical AND gMachine.St.Mode.xAuto;
	iReasonOut.3 := (gMachine.Al.xAlrSafetySystemEStop OR gSafetyController.Alarms.xAlrPrinterEStops) AND gMachine.St.Mode.xManual; //Going out of Manual just for Safety alarms. https://jira.efi.com/browse/CUBE-906

	IF 	iReasonOut > 0	THEN
		IF enPrinterState<>PRINTERGEN_ZERO THEN
			LogOutOfAuto;
		END_IF
		enPrinterState:=PRINTERGEN_ZERO;
	END_IF

	//MachineStates
	gMachine.St.Mode.xZero		:= enPrinterState = PRINTERGEN_ZERO;
	gMachine.St.Mode.xManual	:= enPrinterState = PRINTERGEN_MANUAL;
	gMachine.St.Mode.xAuto		:= enPrinterState = PRINTERGEN_AUTO;
	gMachine.St.Mode.xStartUp	:= enPrinterState = PRINTERGEN_STARTUP;

	// Updated state MANUAL, ZERO OR AUTO
	// This state is used on block, gbelt
	gMachine.St.StateMode:=enPrinterState;

	rsRunBeltOrderManual.SET   := 	gMachine.AutoCmd.xStart;
	rsRunBeltOrderManual.RESET1:= 	gMachine.St.AutoMode.xPause OR
									gMachine.AutoCmd.xStop OR
									gMachine.Al.xAlrSafetySystemEStop OR
									(gLine.Alarms.xCriticalAlarm AND gMachine.Pt.xControlledByLine) OR
									gBelt.AlSummary.xAlarmCritical OR
									gBelt.AlSummary.xAlarmStop OR
									NOT gMachine.St.Mode.xManual;
	rsRunBeltOrderManual();
	g_xRunBeltOrderManual:=rsRunBeltOrderManual.Q1;

	CASE enPrinterState OF

		PRINTERGEN_ZERO:
			gMachine.AutoCmd.iAutoMode:=AUTO_NOT_VALID;

		PRINTERGEN_MANUAL:
			gMachine.AutoCmd.iAutoMode:=AUTO_NOT_VALID;

			//
		PRINTERGEN_AUTO:

			// Normal Cmd
			IF 	NOT gMachine.AlSummary.xAlarmStop AND NOT gMachine.Al.xAlrDisableGoToProduction AND
				// In lab mode doesnt go to production,is just starting belt
				((gMachine.AutoCmd.xStart AND NOT (gMachine.AutoCmd.iAutoMode=AUTO_BYPASS OR gMachine.AutoCmd.iAutoMode=AUTO_LABORATORY) AND NOT gMachine.Pt.xControlledByLine) OR
				(gMachine.commandsSw.xToNormal_GI AND gMachine.St.Blocks.xAnyBlockToPrint)) THEN

					IF gMachine.AutoCmd.iAutoMode<>AUTO_PRODUCTION THEN
						LogAutoInProduction;
					END_IF
					gMachine.AutoCmd.iAutoMode:=AUTO_PRODUCTION;

			END_IF

			//BYPASS
			IF  gMachine.commandsSw.xToByPass_GI OR
				(EDGENEG(gMachine.In.Buttons.xStart) AND NOT tonStartButton.Q AND (gMachine.AutoCmd.iAutoMode=AUTO_STOP) AND NOT gMachine.Pt.xControlledByLine) OR
				EDGEPOS( gMachine.parSw.Dtp.xDoubleLine AND
	            		gMachine.parSw.Dtp.iModeLine1=GC_DTP_BYPASS AND
						gMachine.parSw.Dtp.iModeLine2=GC_DTP_BYPASS) THEN

				IF gMachine.AutoCmd.iAutoMode<>AUTO_BYPASS THEN
					LogAutoInByPass;
				END_IF
				gMachine.AutoCmd.iAutoMode:=AUTO_BYPASS;

			END_IF

			// JAM RECOVERY
			IF  gMachine.commandsSw.xToJamRecovery AND gMachine.Pt.xAllowJamRecovery THEN

				IF gMachine.AutoCmd.iAutoMode<>AUTO_JAMRECOVERY THEN
					LogAutoInJamRecovery;
				END_IF
				gMachine.AutoCmd.iAutoMode:=AUTO_JAMRECOVERY;

			END_IF

			// Laboratory **Conditioins before status OK
			IF  gMachine.commandsSw.xToLaboratory_GI AND gMachine.Pt.xAllowLaboratory THEN
				gMachine.AutoCmd.iAutoMode:=AUTO_LABORATORY;
			END_IF

			// STOP
			iReasonAutoStop.0 := gMachine.AutoCmd.xStop;																						//Stop signal
			iReasonAutoStop.1 := gMachine.AutoCmd.iAutoMode = AUTO_NOT_VALID;																	//Stop by invalid automode
			iReasonAutoStop.2 := gMachine.AutoCmd.iAutoMode <> AUTO_BYPASS AND gMachine.AlSummary.xAlarmStop;									//Stop witohou ByPass with any stop alarm
			iReasonAutoStop.3 := gMachine.AutoCmd.iAutoMode = AUTO_BYPASS AND (gDing.AlSummary.xAlarmStop OR gPhotoCells.AlSummary.xAlarmStop);	//Stop in ByPass with thicknes sensor alarms
			iReasonAutoStop.4 := gMachine.AutoCmd.iAutoMode = AUTO_BYPASS AND																	//Stop in ByPass with TRansVacum stop alarm
								 (gTransVacuum[1].parSw.xActiveOutOfProduction AND gTransVacuum[1].AlSummary.xAlarmStop) OR
								 (gTransVacuum[2].parSw.xActiveOutOfProduction AND gTransVacuum[2].AlSummary.xAlarmStop);

			iReasonAutoStop.5 := gMachine.AutoCmd.iAutoMode = AUTO_BYPASS AND																	//Stop in ByPass with non reference vertical motor alarm
								 (   (gBlock[1].Al.xAlrBarMtrNoRef AND (NOT gBlock[1].In.xTrayIn OR NOT gBlock[1].In.xIclaSensor)) OR
								 (gBlock[2].Al.xAlrBarMtrNoRef AND (NOT gBlock[2].In.xTrayIn OR NOT gBlock[2].In.xIclaSensor))   );

			iReasonAutoStop.6 := ton_JamRecoveryIdle.Q;

			IF  iReasonAutoStop > 0 THEN
				IF gMachine.AutoCmd.iAutoMode<>AUTO_STOP THEN
					iReasonAutoStop_Trigger := iReasonAutoStop;
					iReasonAutoCmdStop_Trigger := iReasonAutoCmdStop;
					LogAutoInStop;
				END_IF
				gMachine.AutoCmd.iAutoMode:=AUTO_STOP;
			END_IF

	END_CASE

	//Define the individual bits for each state
	gMachine.St.AutoMode.xProduction	:= gMachine.AutoCmd.iAutoMode = AUTO_PRODUCTION;
	gMachine.St.AutoMode.xBypass		:= gMachine.AutoCmd.iAutoMode = AUTO_BYPASS;
	gMachine.St.AutoMode.xLaboratory	:= gMachine.AutoCmd.iAutoMode = AUTO_LABORATORY;
	gMachine.St.AutoMode.xStop			:= gMachine.AutoCmd.iAutoMode = AUTO_STOP;
	gMachine.St.AutoMode.xJamRecovery	:= gMachine.AutoCmd.iAutoMode = AUTO_JAMRECOVERY;
	gMachine.St.AutoMode.xProdORLab 	:= gMachine.St.AutoMode.xProduction OR gMachine.St.AutoMode.xLaboratory;
	gMachine.St.AutoMode.xProdORByPass 	:= gMachine.St.AutoMode.xProduction OR gMachine.St.AutoMode.xBypass;

	// State: Pause
	iReasonSetPause.0 := gMachine.commandsSw.xPause_GI;
	iReasonSetPause.1 := EDGEPOS(gMachine.St.AutoMode.xLaboratory);
	iReasonSetPause.2 := EDGEPOS(gMachine.St.Mode.xAuto);
	iReasonSetPause.3 := EDGEPOS(gMachine.In.Buttons.xStart) AND gBelt.states.xRuningBelt;
	srPauseMachine.SET:= iReasonSetPause > 0;

	iReasonResetPause.0 := EDGEPOS(gMachine.St.AutoMode.xBypass);
	iReasonResetPause.1 := EDGEPOS(gMachine.St.AutoMode.xProduction) AND NOT gMachine.Pt.xControlledByLine;
	iReasonResetPause.2 := gMachine.AutoCmd.xStart;
	iReasonResetPause.3 := gMachine.St.AutoMode.xPause AND EDGEPOS(gMachine.In.Buttons.xStart);
	iReasonResetPause.4 := gMachine.St.Mode.xZero;
	iReasonResetPause.5 := gMachine.St.AutoMode.xStop;
	srPauseMachine.RESET1:= iReasonResetPause > 0;
	srPauseMachine();
	gMachine.St.AutoMode.xPause         := srPauseMachine.Q1;

	IF EDGEPOS(gMachine.St.AutoMode.xPause) THEN
		iLastReasonSetPause := iReasonSetPause;
	ELSIF EDGENEG(gMachine.St.AutoMode.xPause) THEN
		iLastReasonResetPause := iReasonResetPause;
	END_IF

	//Machine state to SW, is it used on SW? Or iBlockState?
	CASE gMachine.AutoCmd.iAutoMode OF
		AUTO_PRODUCTION:     gMachine.St.iAutoModeSW:= 1;
		AUTO_BYPASS:         gMachine.St.iAutoModeSW:= 2;
		AUTO_LABORATORY:     gMachine.St.iAutoModeSW:= 3;
		AUTO_JAMRECOVERY:    gMachine.St.iAutoModeSW:= 4;
		AUTO_STOP:           gMachine.St.iAutoModeSW:= 0;
	END_CASE

	tonStartButton(IN:= gMachine.In.Buttons.xStart, PT:= T#1s);

	ton_ZeroMode(IN:= gMachine.St.Mode.xZero, PT:= T#100ms);

	ton_JamRecoveryIdle.IN := gMachine.St.AutoMode.xJamRecovery AND NOT gBelt.states.xRuningBelt;
	ton_JamRecoveryIdle.PT := T#10m;
	ton_JamRecoveryIdle();

END_ACTION
```

#### OrdersPrinter.st - internal commands to all subsytems
```iecst
ACTION OrdersPrinter:

	StatusBlockDetection;
	GeneralAutoCommands;
	GeneralAutoParameters;
	ThicknessControl;
	BlockControl;
	TransportVacuum;
	NonCrashControl;
	CuringLedControl;
	JamDetectControl;
	BeltControl;
	SafetyControl;
	nSensorControl;
	AnalogThicknessControl;
	GeneralControl;
	AncillariesControl;
	EdgeHoldDownControl;
	RemoteCtrl;

END_ACTION

ACTION StatusBlockDetection:

	////////////////////////////////////////////////////////
	// Inputs by comns are auto commands in printer, not all
	//	from kernel: xMute_GI and xReset_GI
	//  from panel: xReset or validate
	////////////////////////////////////////////////////////
	xInCap       		:= TRUE; 	// When all block are capped printer is capped  (AND)
	xInPrint    		:= TRUE;	// When all blocks are printing then is printing (AND)
	xOrderToCapReceived		:= TRUE;
	xOrderToPrintReceived	:= TRUE;
	xGoingToCap  		:= FALSE;
	xGoingToPrint		:= FALSE;
	xCleaning    		:= FALSE;
	xAlarmToEmpyBelt 	:= FALSE;

	FOR iIndexBlock:=GC_FIRST_BLOCK TO gMachine.Pt.CT.iNumBlocks DO
		IF NOT gBlock[iIndexBlock].Status.Position.xInCap THEN
			xInCap:=FALSE;
		END_IF

		IF NOT gBlock[iIndexBlock].Status.Position.xInPrint AND gBlock[iIndexBlock].Status.xEnabledMovements THEN
			xInPrint:=FALSE;
		END_IF

		IF gBlock[iIndexBlock].Status.Position.xGoingToCap THEN
			xGoingToCap:=TRUE;
		END_IF

		IF NOT (gBlock[iIndexBlock].Status.Position.xGoingToCap OR gBlock[iIndexBlock].Status.Position.xInCap) THEN
			xOrderToCapReceived:=FALSE;
		END_IF
		IF NOT (gBlock[iIndexBlock].Status.Position.xGoingToPrint OR gBlock[iIndexBlock].Status.Position.xInPrint) AND gBlock[iIndexBlock].Status.xEnabledMovements THEN
			xOrderToPrintReceived:=FALSE;
		END_IF

		IF gBlock[iIndexBlock].Status.Position.xGoingToPrint THEN
			xGoingToPrint:=TRUE;
		END_IF

		IF gBlock[iIndexBlock].Status.Position.xCleaning THEN
			xCleaning:=TRUE;
		END_IF

		IF gBlock[iIndexBlock].Status.xAlarmToEmptyBelt THEN
			xAlarmToEmpyBelt:=TRUE;
		END_IF

	END_FOR

	//Keeping the signal while the block goes through the next state
	tofMachineCleaning.IN:=xCleaning;
	tofMachineCleaning.PT:=t#150ms;
	tofMachineCleaning();

	gMachine.St.Position.xInCap       	:=	xInCap; 	// When one block is capped printer is capped  (OR)
	gMachine.St.Position.xInPrint    	:=	xInPrint;	// When all blocks are printing then is printing (AND)
	gMachine.St.Position.xGoingToCap  	:=	xGoingToCap;
	gMachine.St.Position.xGoingToPrint	:=	xGoingToPrint;
	gMachine.St.Position.xCleaning    	:=	tofMachineCleaning.Q;
	gMachine.St.Blocks.xBlockAlarmToEmpyBelt 	:= 	xAlarmToEmpyBelt;

	// With these bool are set enPrinterStatesInAuto
	IF gMachine.St.Position.xInCap          THEN enPrinterStatesInAuto:=PRINTER_CAPPED;         END_IF
	IF gMachine.St.Position.xInPrint        THEN enPrinterStatesInAuto:=PRINTER_PRINTING;       END_IF
	IF gMachine.St.Position.xCleaning       THEN enPrinterStatesInAuto:=PRINTER_CLEANING;       END_IF
	IF gMachine.St.Position.xGoingToCap     THEN enPrinterStatesInAuto:=PRINTER_GOING_TO_CAP;   END_IF
	IF gMachine.St.Position.xGoingToPrint	THEN enPrinterStatesInAuto:=PRINTER_GOING_TO_PRINT; END_IF

END_ACTION

ACTION GeneralAutoCommands:

	/////////////////////////////////////////////////////////////////////////////////
	/////////////////////////////////////////////////////////////////////////////////
	//   General auto commads to send block to print or cap from kernel			   //
	/////////////////////////////////////////////////////////////////////////////////
	/////////////////////////////////////////////////////////////////////////////////

	// An edge of commandbooledge must go to cap
	iReasonCap.0 := gMachine.commands.xAllToCap AND (NOT gMachine.St.Position.xInCap);
	iReasonCap.1 := EDGEPOS(gMachine.St.Consent.xUpWithNoConsent);
	iReasonCap.2 := EDGEPOS(gMachine.St.AutoMode.xStop);
	iReasonCap.3 := EDGEPOS(gMachine.St.AutoMode.xBypass);

	iReasonPrint.0 := EDGEPOS(gMachine.commands.xAllToPrint) AND (NOT gMachine.St.Position.xInPrint) AND (gMachine.St.AutoMode.xProdORLab OR gMachine.Pt.xControlledByLine); // An edge of commandbooledge must go to print, if the machine is not stopped
	iReasonPrint.1 := EDGEPOS (gMachine.St.AutoMode.xProduction) AND NOT gMachine.Pt.xControlledByLine; // An edge of auto run must go to print
	iReasonPrint.2 := gMachine.AutoCmd.xStart AND (NOT gMachine.St.Position.xInPrint) AND gMachine.St.AutoMode.xProduction AND NOT gMachine.Pt.xControlledByLine;
	iReasonPrint.3 := EDGEPOS(gMachine.St.Consent.xConsent) AND gMachine.St.Consent.xUpWithNoConsent AND gMachine.St.AutoMode.xProdORLab;
	iReasonPrint.4 := EDGEPOS (gMachine.St.AutoMode.xJamRecovery); // An edge of auto Jam Recovery must go to print

	IF iReasonCap > 0 THEN

		lastReasonCap := iReasonCap;
		gMachine.AutoCmd.xToCap:= TRUE;
		gMachine.AutoCmd.xToPrint:= FALSE;
		iBlockExecutionsOrder := gBlock[1].Status.execTimes;

	ELSIF iReasonPrint > 0 THEN

		lastReasonPrint := iReasonPrint;
		gMachine.AutoCmd.xToCap:= FALSE;
		gMachine.AutoCmd.xToPrint:= TRUE;
		iBlockExecutionsOrder := gBlock[1].Status.execTimes;

	END_IF

	//Fall down orders when received by the blocks
	IF (xOrderToCapReceived) THEN
		gMachine.AutoCmd.xToCap := FALSE;
		iBlockDelay := gBlock[1].Status.execTimes - iBlockExecutionsOrder;
	END_IF
	IF (xOrderToPrintReceived) THEN
		gMachine.AutoCmd.xToPrint := FALSE;
		iBlockDelay := gBlock[1].Status.execTimes - iBlockExecutionsOrder;
	END_IF

	//Ready To print summary variables from blocks
	xMachReadyToPrint := TRUE;
	FOR iIndexBlock:=GC_FIRST_BLOCK TO gMachine.Pt.CT.iNumBlocks DO
		IF gBlock[iIndexBlock].Status.xEnabledMovements AND NOT gBlock[iIndexBlock].Status.Position.xReadyToPrint THEN
			xMachReadyToPrint := FALSE;
		END_IF
	END_FOR

	//When receiving the order to go to print, update the array to avoid going down lower than needed
	IF EDGEPOS(gMachine.AutoCmd.xToPrint) OR EDGEPOS(gMachine.AutoCmd.xToCap) THEN
		gThicknessCtrl.Commands.UpdateAllMatrix:=TRUE;
	END_IF

END_ACTION

ACTION GeneralAutoParameters:

	/////////////////////////////////////////////////////////////////////////////////
	/////////////////////////////////////////////////////////////////////////////////
	//   General PARAMETERS 													   //
	/////////////////////////////////////////////////////////////////////////////////
	/////////////////////////////////////////////////////////////////////////////////

	IF gMachine.Pt.MountedMedia.xDynamicMountedMedia THEN
		IF (gMachine.Pt.MountedMedia.Dynamic.rSpeedMaxMounted = gMachine.Pt.MountedMedia.Dynamic.rSpeedMinMounted) THEN
			//To avoid a divition between 0
			rMountedLimit := 20;
		ELSE
			rMountedLimit := gMachine.Pt.MountedMedia.Dynamic.rMaxOverThickMounted -
			(
			(gBelt.states.rCurrentSpeed - gMachine.Pt.MountedMedia.Dynamic.rSpeedMinMounted) * // Partial of the speed
			(gMachine.Pt.MountedMedia.Dynamic.rMaxOverThickMounted - gMachine.Pt.MountedMedia.Dynamic.rMinOverThickMounted)/ //Range of Overthickness
			(gMachine.Pt.MountedMedia.Dynamic.rSpeedMaxMounted - gMachine.Pt.MountedMedia.Dynamic.rSpeedMinMounted) // Range of speed
			);
		END_IF
		gMachine.St.MountedMedia.rOverThicknessToMounted := LIMIT(gMachine.Pt.MountedMedia.Dynamic.rMinOverThickMounted, rMountedLimit, gMachine.Pt.MountedMedia.Dynamic.rMaxOverThickMounted);
	ELSE
		gMachine.St.MountedMedia.rOverThicknessToMounted := gMachine.parSw.Safety.rMountedPieceOverthickness;
	END_IF

END_ACTION

ACTION ThicknessControl:

	////////////////////////////////////////////////////////////////////////////////
	////////////////////////////////////////////////////////////////////////////////
	/////////////   THICKNESS DETECTION	THICKNESS DETECTION        /////////////////
	/////////////   THICKNESS DETECTION	THICKNESS DETECTION        /////////////////
	////////////////////////////////////////////////////////////////////////////////
	////////////////////////////////////////////////////////////////////////////////

	RejectLength;
	gThicknessCtrl.parameters.Mode  								:= gMachine.St.Mode;
	gThicknessCtrl.parameters.AutoMode								:= gMachine.St.AutoMode;
	gThicknessCtrl.parameters.Belt.rBeltSpeed 						:= gBelt.states.rCurrentSpeed;
	gThicknessCtrl.parameters.ContinuousMedia.MediaData.rThickness	:= gMachine.parSw.Media.rThickness;
	gThicknessCtrl.parameters.ContinuousMedia.MediaData.rMargin		:= gMachine.parSw.rMarginPrint;
	gThicknessCtrl.parameters.Detection.ProductDetect.iMediaFilter	:= gMachine.Pt.iMediaFilter;
	gThicknessCtrl.parameters.rMarginSafePrint						:= gMachine.parSw.Safety.rMarginSafePrint;
	gThicknessCtrl.parameters.iDistanceFromArrayToPd				:= TRUNC(gMachine.Pt.CT.rDistanceThicknesToPD);
	IF gPhotoCells.status.xInstalled THEN
		gThicknessCtrl.parameters.xBlockInProperPrintingPosition 	:= gBlock[1].Status.rMotorPosition <= gPhotoCells.status.rOffsetToReject + gMachine.parSw.Media.rThickness;
	ELSIF gDing.State.xDingInstalled THEN
		gThicknessCtrl.parameters.xBlockInProperPrintingPosition 	:= gBlock[1].Status.rMotorPosition <= gDing.Parameters.rOverThicknessToReject + gMachine.parSw.Media.rThickness;
	END_IF
	gThicknessCtrl.parameters.xBlockInPrint							:= gBlock[1].Status.Position.xInPrint;
	gThicknessCtrl.Inputs.xVirtualMedia 							:= gMachine.Out.xShotLine1 OR gMachine.Out.xShotLine2;

	gThicknessCtrl.Commands.xErrorRst								:= gMachine.AutoCmd.xReset;
	gThicknessCtrl.Commands.xRushProof 								:= gMachine.commandsSw.xRushProof;
	gThicknessCtrl.Commands.xCameraDefectDetected 					:= gMachine.In.xCameraDefectDetected;
	gThicknessCtrl.Commands.xAllowToSetMountedMediaHeigh 			:= NOT gMachine.Pt.xControlledByLine;
	gThicknessCtrl.Commands.xResetMediaBelow						:= gLine.Status = LINE_PREPARING_PRINT;
	gThicknessCtrl.Commands.xReviewIncoherenceArrayAndPd			:= gPhotoCells.status.xInstalled AND (gMachine.Pt.PDSignalTpe=PDCFG_SENSOR);

	gThicknessCtrl.Orders.xDiscardAllMedia							:= gLine.StatusSummary.xEmptyingBelts;

	// If need to add extra height to protect the Printheads, send the information to ThicknessCtrl
	tonRaiseBarsInPause.IN := gMachine.Pt.xProtectPHWithStoppedMediaBended AND gMachine.St.AutoMode.xPause AND gThicknessCtrl.status.MediaPosition.xMediaInside;
	tonRaiseBarsInPause.PT := gMachine.Pt.tiTimeToRaiseBars; //t#5m;
	tonRaiseBarsInPause();
	gMachine.St.xProtectBendedWithPause := tonRaiseBarsInPause.Q;
	IF EDGEPOS(gMachine.St.Consent.xUpWithNoConsent OR gMachine.St.xProtectBendedWithPause) AND NOT gTransVacuum[1].Status.xInstalled THEN
		gThicknessCtrl.Commands.xAddSafetyMarginToHeight := TRUE;
	END_IF

END_ACTION

ACTION BlockControl:

	///////////////////////////////////////////////////////////////////////////////////
	///////////////////////////////////////////////////////////////////////////////////
	/////////////   BLOCK BLOCK BLOCK BLOCK BLOCK BLOCK BLOCK      ////////////////////
	/////////////   BLOCK BLOCK BLOCK BLOCK BLOCK BLOCK BLOCK      ////////////////////
	///////////////////////////////////////////////////////////////////////////////////
	///////////////////////////////////////////////////////////////////////////////////

	//Up bars by bent tile
	tonDelayToSafetyPos.IN:= gThicknessCtrl.status.MediaPosition.xMediaBelowMachine AND NOT gBelt.states.xRuningBelt AND
							((gMachine.Pt.xProtectPHWithStoppedMediaBended AND gMachine.St.AutoMode.xProduction) OR (gMachine.Pt.xProtectPHForBlowersRunning AND gTransVacuum[1].Status.State = TRANSVAC_CONTROLLING));
	tonDelayToSafetyPos.PT:= T#1m;
	tonDelayToSafetyPos();

	srUpBarsToSafePos.SET1	:= 	EDGEPOS(tonDelayToSafetyPos.Q);
	srUpBarsToSafePos.RESET	:= 	NOT gThicknessCtrl.status.MediaPosition.xMediaBelowMachine  OR
								(EDGEPOS(gMachine.St.Consent.xConsent) OR EDGEPOS(gBelt.commands.xRunBelt));
	srUpBarsToSafePos();

	gMachine.AutoCmd.xToSafePosition := srUpBarsToSafePos.Q1;

	// Reason Move Bars to PrePrinting Position
	tonProtecPHBlowers.IN :=	gMachine.Pt.xProtectPHForBlowersRunning AND
								NOT gThicknessCtrl.status.MediaPosition.xMediaInside AND
								NOT gThicknessCtrl.status.MediaPosition.xVirtualMediaInside AND
								(gTransVacuum[1].Status.State = TRANSVAC_CONTROLLING OR gMachine.St.AutoMode.xPause) AND
								gMachine.St.Mode.xAuto AND gMachine.St.Position.xInPrint AND
								NOT gMachine.Pt.xControlledByLine AND
								(NOT gMachine.parSw.Remote.xSendingJob OR NOT gMachine.Pt.xControlledRemotely);
	tonProtecPHBlowers.PT := t#20s;
	tonProtecPHBlowers();

	// 1 sec after receiving the SendingJob signal, it is reseted
	tonResetSendingJob.IN := gMachine.parSw.Remote.xSendingJob;
	tonResetSendingJob.PT := t#1s;
	tonResetSendingJob();
	IF tonResetSendingJob.Q THEN
		gMachine.parSw.Remote.xSendingJob := FALSE;
	END_IF

	iReasonForcePreprintingPos.0 := tonProtecPHBlowers.Q;
	iReasonForcePreprintingPos.1 := gLine.Orders.Preprinting;
	iReasonForcePreprintingPos.2 := gMachine.AutoCmd.xToSafePosition;
	iReasonForcePreprintingPos.3 := gLine.StatusSummary.xEmptyingBelts;
	iReasonForcePreprintingPos.4 := gEdgeHoldDown.parSw.xEnable AND NOT gEdgeHoldDown.status.xAdjustedToMedia;
	iReasonForcePreprintingPos.5 := gMachine.St.AutoMode.xJamRecovery;
	iReasonForcePreprintingPos.6 := gThicknessCtrl.status.MediaPosition.xMountedMediaInside;
	iReasonForcePreprintingPos.7 := gLine.StatusSummary.xCleaningBelt;

	// Registering PrePrintingPos
	IF iPrevReasonForcePreprintingPos <> iReasonForcePreprintingPos THEN
		LogPrePrintingPos;
	END_IF
	iPrevReasonForcePreprintingPos := iReasonForcePreprintingPos;

	xForcePreprintingPos := (iReasonForcePreprintingPos>0);

	FOR iIndexBlock:=GC_FIRST_BLOCK TO gMachine.Pt.CT.iNumBlocks DO

		//NOTE: Sw and Slow information is sent to the Block in MachineSlow >> OrdersPrinterSlow

		// It sends blocks to pirnting state because is required by mode active printer
		gBlock[iIndexBlock].commands.StateMode  := gMachine.St.StateMode;
		gBlock[iIndexBlock].commands.Mode  		:= gMachine.St.Mode;
		gBlock[iIndexBlock].commands.AutoMode	:= gMachine.St.AutoMode;
		IF gMachine.AutoCmd.xToCap THEN  gBlock[iIndexBlock].commands.xToCap := TRUE; END_IF //This is to allow individual orders
		IF gMachine.AutoCmd.xToPrint THEN  gBlock[iIndexBlock].commands.xToPrint := TRUE; END_IF //This is to allow individual orders
		gBlock[iIndexBlock].commands.xReset		:= gMachine.AutoCmd.xReset;
		gBlock[iIndexBlock].commands.xMute		:= gMachine.AutoCmd.xMuteAlarms;
		gBlock[iIndexBlock].commands.xCleanStop	:= gMachine.AlSummary.xAlrSafetySystemGeneral;
		gBlock[iIndexBlock].commands.xForcePreprintingPos := xForcePreprintingPos;

		gBlock[iIndexBlock].parameters.Motor.rPrintPosition		:= gThicknessCtrl.status.Heigh.rMaxHeigh[iIndexBlock];
		gBlock[iIndexBlock].parameters.xLeftHandMachine			:= gMachine.Pt.xLeftHandMachine;
		gBlock[iIndexBlock].parameters.xRightHandMachine		:= gMachine.Pt.xRightHandMachine;
		gBlock[iIndexBlock].parameters.xMediaBelow				:= NOT gThicknessCtrl.status.Belt.xBeltEmpty;
		gBlock[iIndexBlock].parameters.xPrinterKeyMaintenanceActivated := gSafetyController.Inputs.xPrinterMaintenanceKey AND gSafetyController.Parameters.xInstalled;

	END_FOR

END_ACTION

ACTION TransportVacuum:

	///////////////////////////////////////////////////////////////////////////////////
	///////////////////////////////////////////////////////////////////////////////////
	/////////////   TRANSPORT VACUUM   TRANSPORT VACUUM     ///////////////////////////
	/////////////   TRANSPORT VACUUM   TRANSPORT VACUUM     ///////////////////////////
	///////////////////////////////////////////////////////////////////////////////////
	///////////////////////////////////////////////////////////////////////////////////

	FOR usiIndex:=1 TO gMachine.Pt.CT.iNumTransVacuum BY 1 DO
		OrdersToTransVacuum;
	END_FOR

END_ACTION

ACTION NonCrashControl:

	///////////////////////////////////////////////////////////////////////////////////
	///////////////////////////////////////////////////////////////////////////////////
	///////////   NON CRASH   NON CRASH   NON CRASH   NON CRASH    ////////////////////
	///////////   NON CRASH   NON CRASH   NON CRASH   NON CRASH    ////////////////////
	///////////////////////////////////////////////////////////////////////////////////
	///////////////////////////////////////////////////////////////////////////////////

	IF gNonCrash[1].Status.xInstalled THEN

		gNonCrash[1].Parameters.Mode := gMachine.St.Mode;
		gNonCrash[1].Parameters.AutoMode := gMachine.St.AutoMode;

		gNonCrash[1].Parameters.rSpeedSetPoint := gBelt.parameters.rSetPointSpeed;

		gNonCrash[1].Commands.xRun := gBelt.states.xRuningBelt;
		gNonCrash[1].Commands.xMute := gMachine.AutoCmd.xMuteAlarms;
		gNonCrash[1].Commands.xReset := gMachine.AutoCmd.xReset;

		//Safety Alarm Summary
		gNonCrash[1].Commands.xExternalSafetyStop := gMachine.AlSummary.xAlrSafetySystemGeneral;

	END_IF

END_ACTION

ACTION CuringLedControl:

	///////////////////////////////////////////////////////////////////////////////////
	///////////////////////////////////////////////////////////////////////////////////
	/////////// CURING LED    CURING LED    CURING LED    CURING LED   ////////////////
	/////////// CURING LED    CURING LED    CURING LED    CURING LED   ////////////////
	///////////////////////////////////////////////////////////////////////////////////
	///////////////////////////////////////////////////////////////////////////////////
	FOR iIndexCuringBar:=1 TO MAX_LAST_CURING_LED DO

		iReasonRunNitrogenFlow.0 := (gBelt.states.rCurrentSpeed>=gCuringLed[iIndexCuringBar].Parameters.rMinCureSpeed) AND
									(gMachine.St.AutoMode.xProdORLab OR gMachine.St.AutoMode.xJamRecovery) AND
									NOT gMachine.St.Position.xCleaning;
		iReasonRunNitrogenFlow.1 := (gBelt.states.rCurrentSpeed>=gCuringLed[iIndexCuringBar].Parameters.rMinCureSpeed) AND gLine.StatusSummary.xControlStopping;
		iReasonRunNitrogenFlow.2 := gLine.StatusSummary.xEmptyingBelts;
		iReasonRunNitrogenFlow.3 := gLine.StatusSummary.xPrinting;

		IF gCuringLed[iIndexCuringBar].Parameters.xInstalled THEN
			gCuringLed[iIndexCuringBar].Parameters.Mode 			:= gMachine.St.Mode;
			gCuringLed[iIndexCuringBar].Parameters.AutoMode 		:= gMachine.St.AutoMode;

			//Evaluating media is in curing led bar position
			xMediaInLedPosition := FALSE;
			IF gCuringLed[iIndexCuringBar].Parameters.CuringApplicationType = CURING_APP_WHITE THEN
				xMediaInLedPosition := (gThicknessCtrl.status.MediaPosition.L1.White.xMediaInLedPosition OR gThicknessCtrl.status.MediaPosition.L2.White.xMediaInLedPosition);

			ELSIF gCuringLed[iIndexCuringBar].Parameters.CuringApplicationType = CURING_APP_COLOR THEN
				xMediaInLedPosition := (gThicknessCtrl.status.MediaPosition.L1.Color.xMediaInLedPosition OR gThicknessCtrl.status.MediaPosition.L2.Color.xMediaInLedPosition);

			ELSIF gCuringLed[iIndexCuringBar].Parameters.CuringApplicationType = CURING_APP_PRIMER THEN
				xMediaInLedPosition := (gThicknessCtrl.status.MediaPosition.L1.Primer.xMediaInLedPosition OR gThicknessCtrl.status.MediaPosition.L2.Primer.xMediaInLedPosition);
			END_IF

			//Defining which curing led bar have to cure always when in printing (related to jam recovery/empty belt processes when only one the several curing led bars have to cure
			IF iIndexCuringBar=gMachine.Pt.Hw.iMaxCuringLedBars THEN
				xCuringDesired[iIndexCuringBar] := gBlock[1].Status.Position.xInPrint;
			ELSE
				xCuringDesired[iIndexCuringBar] := gThicknessCtrl.parameters.xBlockInProperPrintingPosition;
			END_IF

			//Commands
			gCuringLed[iIndexCuringBar].Commands.PowerOn 				:= NOT gSafetyController.Alarms.xCriticalAlarm;
			gCuringLed[iIndexCuringBar].Commands.Mute 				:= gMachine.AutoCmd.xMuteAlarms;
			gCuringLed[iIndexCuringBar].Commands.Reset 				:= gMachine.AutoCmd.xReset;

			IF gCuringLed[iIndexCuringBar].Parameters.xEnabled THEN
				gCuringLed[iIndexCuringBar].Commands.RunCuring 			:= 	xMediaInLedPosition AND
																			(gBelt.states.rCurrentSpeed>=gCuringLed[1].Parameters.rMinCureSpeed) AND
																			gBelt.states.xRuningBelt AND //This condition seems repeated but just for safety
																			(xCuringDesired[iIndexCuringBar] OR gMachine.St.AutoMode.xJamRecovery) AND
																			gMachine.St.Mode.xAuto; //This condition was required in DELOREAN-442

				gCuringLed[iIndexCuringBar].Commands.xDropPower	 		:= gLine.StatusSummary.xEmptyingBelts OR NOT gThicknessCtrl.parameters.xBlockInProperPrintingPosition OR gMachine.St.AutoMode.xJamRecovery;
				gCuringLed[iIndexCuringBar].Commands.xRunNitrogenFlow 	:= (iReasonRunNitrogenFlow>0);
				gCuringLed[iIndexCuringBar].Commands.xUpdateTempValues 	:= gPLC.Internal.Blink_10s.Out;
			END_IF

		END_IF
	END_FOR

END_ACTION

ACTION JamDetectControl:

	/////////////////////////////////////////////////////////////////////////////////
	/////////////////////////////////////////////////////////////////////////////////
	/////////////   JAM DETECT	JAM DETECT	JAM DETECT	JAM DETECT	/////////////////
	/////////////   JAM DETECT	JAM DETECT	JAM DETECT	JAM DETECT	/////////////////
	/////////////////////////////////////////////////////////////////////////////////
	/////////////////////////////////////////////////////////////////////////////////

	IF gMachine.St.iJamDevices > 0 THEN
		OrdersToJamVibration;
	END_IF

	//Wait finish JamTesting to start belt
	xStopBeltJamTesting :=	gMachine.parSw.xJamDetectEnable AND
							gMachine.St.AutoMode.xProduction AND
							(gBlock[1].Status.PositionState = BLOCKP_IN_PRINT OR gBlock[2].Status.PositionState = BLOCKP_IN_PRINT) AND
							(gJamDetect[1].Status = JAMVIB_TESTING OR gJamDetect[2].Status = JAMVIB_TESTING);

END_ACTION

ACTION BeltControl:

	///////////////////////////////////////////////////////////////////////////////////
	///////////////////////////////////////////////////////////////////////////////////
	/////////////   BELT  BELT  BELT  BELT  BELT  BELT  BELT  BELT  ///////////////////
	/////////////   BELT  BELT  BELT  BELT  BELT  BELT  BELT  BELT  ///////////////////
	///////////////////////////////////////////////////////////////////////////////////
	///////////////////////////////////////////////////////////////////////////////////

	IF gMachine.St.Position.xCleaning AND (gMachine.St.xMediaDetected) AND NOT gMachine.St.AutoMode.xBypass THEN
		xStopBeltWhileCleaning:= TRUE;
	ELSIF NOT gMachine.St.Mode.xAuto OR NOT gMachine.St.Position.xCleaning THEN
		xStopBeltWhileCleaning:= FALSE;
	END_IF

	srStopBeltNoImage.SET1 := gMachine.Al.Warning.xNotLoadedImage AND NOT gMachine.Pt.xControlledByLine;
	srStopBeltNoImage.RESET := NOT gMachine.St.Mode.xAuto OR NOT gMachine.St.Position.xInPrint OR NOT gMachine.Al.Warning.xNotLoadedImage;
	srStopBeltNoImage();

	iReasonStopBeltAuto.0 := gMachine.AlSummary.xAlarmStop AND NOT gMachine.St.AutoMode.xBypass;
	iReasonStopBeltAuto.1 := gMachine.Al.Alarm.xAlarmMountedPiece;
	iReasonStopBeltAuto.2 := xStopBeltWhileCleaning;
	iReasonStopBeltAuto.3 := gMachine.AlSummary.xAlarmStop AND gMachine.Pt.xControlledByLine;
	iReasonStopBeltAuto.4 := xStopBeltJamTesting;
	xSignalsStopBeltAuto:= 	iReasonStopBeltAuto > 0;

	xAlarmsStopBeltRun:= 	srStopBeltNoImage.Q1 OR gMachine.Al.Alarm.xAlarmNotInPrintPosition;

	//Not stop de belt while the user raises the bars
	IF gMachine.commands.xAllToCap THEN
		xUserRaisesBlocks := TRUE;
	END_IF
	IF NOT gMachine.St.AutoMode.xProduction OR EDGEPOS(gMachine.St.Position.xInPrint) THEN
		xUserRaisesBlocks := FALSE;
	END_IF

	IF EDGEPOS(gMachine.St.Consent.xUpWithNoConsent) THEN
		xMachineRaisesBlock := TRUE;
	END_IF
	IF NOT gMachine.St.AutoMode.xProduction OR EDGEPOS(gMachine.St.Position.xInPrint) THEN
		xMachineRaisesBlock := FALSE;
	END_IF

	iReasonOrdersRunBeltProduction.0 := gMachine.St.Position.xInPrint;
	iReasonOrdersRunBeltProduction.1 := (xUserRaisesBlocks OR xMachineRaisesBlock) AND NOT gMachine.Pt.xControlledByLine;
	iReasonOrdersRunBeltProduction.2 := gMachine.St.xBeltRunPrevToClean AND (gMachine.St.Position.xGoingToPrint OR gMachine.St.Position.xCleaning);
	xOrdersRunBeltNormal := iReasonOrdersRunBeltProduction > 0 ;

	IF EDGEPOS((gPhotoCells.status.xInPosition) AND gMachine.St.AutoMode.xProdORLab) THEN
		iReasonORunBeltPhoto := TRUE;
	ELSIF NOT gMachine.St.Mode.xAuto OR EDGENEG(gMachine.St.AutoMode.xProdORLab) THEN
		iReasonORunBeltPhoto := FALSE;
	END_IF

	xRunBeltNormal:= gMachine.St.AutoMode.xProduction AND
					NOT xAlarmsStopBeltRun AND
					xOrdersRunBeltNormal AND
					(NOT gPhotoCells.parameters.xInstall OR iReasonORunBeltPhoto);

	xRunBeltByLine := (gMachine.Pt.xControlledByLine AND gMachine.commands.xRunBelt AND NOT xAlarmsStopBeltRun);

	xRunBeltByPass := gMachine.St.AutoMode.xBypass; //Start bypass with run belt order. Stopped by pause when desired

	xRunBeltLab:= gMachine.St.AutoMode.xLaboratory AND NOT xAlarmsStopBeltRun;

	xRunBeltToBeCleaned := (gMachine.Pt.Clean.xCleanBeltForUv AND gMachine.commands.xRunBelt AND NOT xAlarmsStopBeltRun);

	//Consider PAUSE just with the final order. Not in the 3 previous
	g_xRunBeltOrderAuto	:= (xRunBeltNormal OR xRunBeltByPass OR xRunBeltLab OR xRunBeltByLine OR xRunBeltToBeCleaned) AND NOT xSignalsStopBeltAuto AND ((NOT gMachine.St.AutoMode.xPause AND NOT gMachine.Pt.xControlledByLine) OR gMachine.Pt.xControlledByLine);

	//Writing belt commands
	gBelt.commands.xMute      	:= gMachine.AutoCmd.xMuteAlarms;
	gBelt.commands.xReset     	:= gMachine.AutoCmd.xReset;
	gBelt.commands.Mode			:= gMachine.St.Mode;
	gBelt.commands.AutoMode		:= gMachine.St.AutoMode;
	gBelt.commands.xRunBelt	  	:= g_xRunBeltOrderAuto OR g_xRunBeltOrderManual;
	gBelt.commands.xJogBelt	  	:= gMachine.St.Mode.xAuto AND (gMachine.St.AutoMode.xStop OR (gMachine.St.AutoMode.xJamRecovery AND gMachine.St.Remote.xReadyToJogInJamRecovery)) AND gTransVacuum[1].Status.Blower.xMoving AND gMachine.In.xRemoteJog;
	gBelt.commands.xUseJogAccDecc := gMachine.St.AutoMode.xJamRecovery;
	gBelt.commands.xUseSoftDeceleration := gMachine.Pt.xControlledByLine AND (gMachine.St.Mode.xManual OR (NOT gMachine.Al.Alarm.xAlarmMountedPiece AND NOT gLine.Alarms.xCriticalAlarm)); //[RGP] Applies only for machine controlled by line at the moment

	//Safety Alarm Summary
	gBelt.commands.xExternalSafetyStop := gMachine.AlSummary.xAlrSafetySystemGeneral;

	//Printer gives consent to belt here
	gBelt.commands.xConsentBelt:= 	gMachine.St.AutoMode.xLaboratory OR
									(NOT gMachine.Pt.xControlledByLine AND gMachine.St.Consent.xConsent AND NOT gMachine.St.Consent.xUpWithNoConsent) OR
									(gMachine.Pt.xControlledByLine AND NOT gLine.Alarms.xCriticalAlarm);

END_ACTION

ACTION SafetyControl:

	//Safety
	gSafetyController.Commands.xReset := gMachine.AutoCmd.xReset;

END_ACTION

ACTION nSensorControl:

	IF gPhotoCells.status.xInstalled THEN
		tonResetCommandIcla.IN := gMachine.AutoCmd.xReset;
		tonResetCommandIcla.PT := T#2S ;
		tonResetCommandIcla();

		//Writing 3 Lasers COMMANDS
		gPhotoCells.commands.xResetMotor			:=	tonResetCommandIcla.Q OR EDGENEG(gMachine.AlSummary.xAlarmCritical); //NOZOMITWO-944: Adding non critical alarm condition to reset motor
		gPhotoCells.commands.xErrorRst				:=	gMachine.AutoCmd.xReset;
		gPhotoCells.commands.xMute					:=	gMachine.AutoCmd.xMuteAlarms;
		gPhotoCells.commands.Mode					:=	gMachine.St.Mode;
		gPhotoCells.commands.AutoMode				:=	gMachine.St.AutoMode;
		gPhotoCells.commands.xCancelAlignmentCheck	:= 	gMachine.St.Position.xGoingToPrint OR NOT gMachine.St.Mode.xAuto OR gLine.StatusSummary.xEmptyingBelts OR gMachine.St.CleaningBelt.xCleaningProcessOnGoing;
		gPhotoCells.commands.xCheckMounted			:= 	(gBelt.states.xRuningBelt OR gBelt.commands.xRunBelt) AND
														(NOT gMachine.St.AutoMode.xBypass OR ((*ByPassConditions>>*) gPhotoCells.parameters.xEnableMountedAlrByPass)) AND
														(NOT gMachine.Pt.xControlledByLine OR ((*LineConditions>>*) NOT gMachine.St.CleaningBelt.xCleaningProcessOnGoing ));
		gPhotoCells.commands.xRecordMaxPosition		:= (gBelt.states.xRuningBelt OR gBelt.commands.xRunBelt);
		gPhotoCells.commands.xMountedMediaInside := gThicknessCtrl.status.MediaPosition.xMountedMediaInside;

		//Writing photocells parameters
		gPhotoCells.parameters.rMediaThickness	:=	gThicknessCtrl.status.Heigh.rMediaThickness;
		gPhotoCells.parameters.rMarginPrint	:=	gMachine.parSw.rMarginPrint;
		gPhotoCells.parameters.rPrePrintPosition := gBlock[1].parameters.rPrePrintingPos;
		gPhotoCells.parameters.xHomingEnabled := gTransVacuum[1].Status.xAtSpeed OR NOT gTransVacuum[1].Status.xInstalled;

	END_IF

END_ACTION

ACTION AnalogThicknessControl:

	///////////////////////////////////////////////////////////////////////////////////
	///////////////////////////////////////////////////////////////////////////////////
	/////////////   DING   DING   DING   DING   DING   DING   DING  ///////////////////
	/////////////   DING   DING   DING   DING   DING   DING   DING  ///////////////////
	///////////////////////////////////////////////////////////////////////////////////
	///////////////////////////////////////////////////////////////////////////////////

	IF gDing.State.xDingInstalled THEN
		gDing.Commands.xMute		:= gMachine.AutoCmd.xMuteAlarms;
		gDing.Commands.xErrorRst	:= gMachine.AutoCmd.xReset;
		gDing.Commands.Mode			:= gMachine.St.Mode;
		gDing.Commands.AutoMode		:= gMachine.St.AutoMode;
		gDing.Commands.xMountedMediaInside := gThicknessCtrl.status.MediaPosition.xMountedMediaInside;

		gDing.In.xAnyCarriageProductDetect := gMachine.St.ProductDetect.xProductDetectL1 OR gMachine.St.ProductDetect.xProductDetectL2;
		gDing.Parameters.rMediaThickness := gMachine.parSw.Media.rThickness;
		gDing.Parameters.rMarginPrint	:=	gMachine.parSw.rMarginPrint;
		gDing.Parameters.rOverThicknessToMounted := gMachine.St.MountedMedia.rOverThicknessToMounted;
		gDing.Parameters.rMarginSafePrint := gMachine.parSw.Safety.rMarginSafePrint;
	END_IF

END_ACTION

ACTION GeneralControl:

	//////////Cooling PC Cabinet///////////
	gMachine.Out.xCoolingPCStart := TRUE; //ALX - For the moment is On avery time, its posible control this but its necesary check in machine

	//Removing the commands
	gMachine.commands.xAllToCap:=FALSE;
	gMachine.commands.xAllToPrint:=FALSE;
	gMachine.commands.xStop:=FALSE;

	//Command to abort job for SW
	IF NOT gMachine.St.xRobotReadyToPrint THEN
		gMachine.St.xAbortJobRequest:=FALSE;

	ELSIF gMachine.AlSummary.xAnyAlarm THEN
		gMachine.St.xAbortJobRequest:=TRUE;
	END_IF

END_ACTION

ACTION AncillariesControl:

	///////////////////////////////////////////////////////////////////////////////////
	///////////////////////////////////////////////////////////////////////////////////
	/////////////   ANCILLARIES ANCILLARIES ANCILLARIES ANCILLARIES ///////////////////
	/////////////   ANCILLARIES ANCILLARIES ANCILLARIES ANCILLARIES ///////////////////
	///////////////////////////////////////////////////////////////////////////////////
	///////////////////////////////////////////////////////////////////////////////////

	gStacker.Orders.xRejectSheet := gThicknessCtrl.Outputs.xReject;

END_ACTION

ACTION OrdersToTransVacuum:

	IF NOT gTransVacuum[usiIndex].Status.xInstalled THEN
		RETURN;
	END_IF

	//Avoid memory when not in manual
	IF gMachine.St.StateMode <> PRINTERGEN_MANUAL THEN
		gTransVacuum[usiIndex].OrdersSw.xRunManual := FALSE;
	END_IF

	//DELOREAN-2585
	//Service has asked to active vacuum at full power when homing photocell's motor.
	//May be disactivated when homing process has finished or via HMI
	IF EDGEPOS(gPhotoCells.status.xReferencing) THEN
		gTransVacuum[1].OrdersSw.xRunManual := TRUE;
		gTransVacuum[1].parSw.rManSetPoint := 100.0;
	END_IF
	IF EDGEPOS(gPhotoCells.status.xReferenced) THEN
		gTransVacuum[1].OrdersSw.xRunManual := FALSE;
	END_IF

	//Applying coefficient to vacuum pressure setpoint depending on line state
	IF gMachine.Pt.xControlledByLine THEN
		IF gLine.StatusSummary.xEmptyingBelts THEN
			rCoef := 1.3;
		ELSIF ((gLine.StatusSummary.xPausing AND gThicknessCtrl.status.Belt.xBeltEmpty) OR gLine.StatusSummary.xCleaning) THEN
			rCoef := 0;
		ELSIF gLine.StatusSummary.xPrinting THEN
			rCoef := 1.0;
		END_IF

	ELSE
		rCoef := 1.0;
	END_IF

	gTransVacuum[1].Parameters.rVacPressureSetPointPerc := LIMIT(gTransVacuum[1].Parameters.rMinVacPressureSetPointPerc, (gTransVacuum[1].parSw.rVacPressureSetPointPerc*rCoef), 100);

	//If needed to send parameters to other TransVacuum
	IF NOT gMachine.Pt.Vacuum.xTransVacuumIndependenParams AND usiIndex>1 THEN
		gTransVacuum[usiIndex].OrdersSw.xRunManual					:= gTransVacuum[1].OrdersSw.xRunManual;
		gTransVacuum[usiIndex].parSw.xActiveOutOfProduction 		:= gTransVacuum[1].parSw.xActiveOutOfProduction;
		gTransVacuum[usiIndex].parSw.rManSetPoint					:= gTransVacuum[1].parSw.rManSetPoint;
		gTransVacuum[usiIndex].Parameters.rStartUpDutyCycle			:= gTransVacuum[1].Parameters.rStartUpDutyCycle;
		gTransVacuum[usiIndex].Parameters.rVacPressureSetPointPerc	:= gTransVacuum[1].Parameters.rVacPressureSetPointPerc;
	END_IF

	gTransVacuum[usiIndex].Commands.xMute := gMachine.AutoCmd.xMuteAlarms;
	IF gMachine.AutoCmd.xReset OR xEdgeSafety THEN
		gTransVacuum[usiIndex].Commands.xReset := TRUE;
	END_IF
	gTransVacuum[usiIndex].Commands.xRunJamRecovery := gMachine.St.AutoMode.xJamRecovery;

	IF EDGE(gMachine.St.Position.xGoingToPrint AND gMachine.St.AutoMode.xProdORLab) THEN
		xStartVacuumWhileGoingDown := TRUE;
	END_IF
	IF gBelt.states.xRuningBelt OR gMachine.St.Position.xGoingToCap OR gMachine.St.Position.xInCap THEN
		xStartVacuumWhileGoingDown := FALSE;
	END_IF

	xReasonRunVacuumProduction.0 := gBelt.states.xOrderRuning;
	xReasonRunVacuumProduction.1 := gThicknessCtrl.status.MediaPosition.xMediaInside AND gMachine.St.AutoMode.xProdORLab;
	xReasonRunVacuumProduction.2 := gMachine.Pt.Vacuum.xStartBlowerGoingToPrint AND xStartVacuumWhileGoingDown;
	gTransVacuum[usiIndex].Commands.xRunProduction := xReasonRunVacuumProduction > 0 ;

	//Safety Alarm Summary
	gTransVacuum[usiIndex].Parameters.xExternalSafetyStop := gMachine.AlSummary.xAlrSafetySystemGeneral OR gSafetyController.Alarms.xAlrBlowersEnclosureSwitchOff;

	gTransVacuum[usiIndex].Parameters.AutoMode := gMachine.St.AutoMode;
	gTransVacuum[usiIndex].Parameters.Mode := gMachine.St.Mode;
	gTransVacuum[usiIndex].Parameters.xBeltRunning := gBelt.states.xOrderRuning;

	//In remote controlled machines, Commands.xRunByLine is used to allow remote blowers running
	IF gMachine.Pt.xControlledRemotely THEN
		iReasonRunBlowerRemote.0 := gMachine.St.AutoMode.xStop AND gMachine.commands.Remote.xStartBlowers;
		iReasonRunBlowerRemote.1 := gMachine.St.AutoMode.xBypass;
		gTransVacuum[usiIndex].Commands.xRunByRemote := gMachine.St.Mode.xAuto AND iReasonRunBlowerRemote>0;
	END_IF

END_ACTION

ACTION EdgeHoldDownControl:
	IF gEdgeHoldDown.status.xInstalled THEN
		//Writing commands
		gEdgeHoldDown.commands.xErrorRst			:= tonResetCommandIcla.Q OR EDGENEG(gMachine.AlSummary.xAlarmCritical); //NOZOMITWO-944: Adding non critical alarm condition to reset motor
		gEdgeHoldDown.commands.xErrorRst			:= gMachine.AutoCmd.xReset;
		gEdgeHoldDown.commands.xMute				:= gMachine.AutoCmd.xMuteAlarms;
		gEdgeHoldDown.commands.Mode					:= gMachine.St.Mode;
		gEdgeHoldDown.commands.AutoMode				:= gMachine.St.AutoMode;

		//Writing parameters
		gEdgeHoldDown.parameters.rBarsHeighSp 		:= gMachine.parSw.Media.rThickness + gMachine.parSw.rMarginPrint;
		gEdgeHoldDown.parameters.rWidthSp 			:= gMachine.parSw.Media.rWidth;
		gEdgeHoldDown.parameters.rBlockPosition		:= gBlock[1].Status.rMotorPosition;

		gPairedMotors[1].commands.xMute				:= gMachine.AutoCmd.xMuteAlarms;
		gPairedMotors[1].commands.Mode				:=	gMachine.St.Mode;
		gPairedMotors[1].commands.xErrorRst			:=	gMachine.AutoCmd.xReset;
		gPairedMotors[1].commands.xResetMotor		:=	tonResetCommandIcla.Q OR EDGENEG(gMachine.AlSummary.xAlarmCritical);

		gPairedMotors[2].commands.xMute				:= gMachine.AutoCmd.xMuteAlarms;
		gPairedMotors[2].commands.Mode				:=	gMachine.St.Mode;
		gPairedMotors[2].commands.xErrorRst			:=	gMachine.AutoCmd.xReset;
		gPairedMotors[2].commands.xResetMotor		:=	tonResetCommandIcla.Q OR EDGENEG(gMachine.AlSummary.xAlarmCritical);

	END_IF

END_ACTION

ACTION OrdersToJamVibration:

	IF NOT gMachine.parSw.xJamDetectEnable THEN
		FOR	usiIndex:=1 TO gMachine.St.iJamDevices DO gJamDetect[usiIndex].Parameters.xJamEnabled := FALSE; END_FOR
		RETURN;
	END_IF

	FOR iIndexBlock := 1  TO gMachine.Pt.CT.iNumBlocks DO

		FOR usiIndex:=1 TO gMachine.St.iJamDevices DO

			//JamDevice in proper block
			IF gJamDetect[usiIndex].Parameters.iBlock = iIndexBlock THEN

				//Send common data
				gJamDetect[usiIndex].Parameters.xJamEnabled	:= gMachine.parSw.xJamDetectEnable;
				gJamDetect[usiIndex].Commands.xReset 		:= gMachine.AutoCmd.xReset;
				gJamDetect[usiIndex].Commands.xMuteAlarms	:= gMachine.AutoCmd.xMuteAlarms;

				//Send order to work
				IF  gMachine.St.Mode.xAuto AND NOT gBlock[iIndexBlock].commands.xStartToCleanOrder THEN

					gJamDetect[usiIndex].Commands.xStart := TRUE;

				ELSE

					gJamDetect[usiIndex].Commands.xStart := FALSE;

				END_IF

				//Pause order
				gJamDetect[usiIndex].Commands.xPause :=	gBlock[iIndexBlock].Status.PositionState = BLOCKP_CLEANING OR
														gBlock[iIndexBlock].Status.PositionState = BLOCKP_GOING_TO_PRINT OR
														(gBlock[iIndexBlock].Status.PositionState <> BLOCKP_IN_PRINT AND gJamDetect[usiIndex].Commands.xStart) OR
														(gBlock[iIndexBlock].Status.PositionState = BLOCKP_IN_PRINT AND NOT gBelt.commands.xRunBelt AND NOT gBlock[iIndexBlock].commands.xStartToCleanOrder);

			END_IF

		END_FOR
	END_FOR

END_ACTION

ACTION RejectLength:

	//Calculate the distance of the devices between the Printer and the Stacker
	IF NOT gDryerAnc.Parameters.xInstalled AND NOT gOverVarnish.Parameters.xInstalled THEN
		iDistanceMiddleDevices := 0;
	ELSIF gDryerAnc.Parameters.xInstalled AND NOT gOverVarnish.Parameters.xInstalled THEN
		IF gBelt.states.rCurrentSpeed > 70.0 THEN
			iDistanceMiddleDevices := REAL_TO_INT((gDryerAnc.Parameters.Hw.rDryerLength/10) - (2*(gBelt.states.rCurrentSpeed - 70.0)));
		ELSE
			iDistanceMiddleDevices := REAL_TO_INT(gDryerAnc.Parameters.Hw.rDryerLength/10);
		END_IF
	ELSIF NOT gDryerAnc.Parameters.xInstalled AND gOverVarnish.Parameters.xInstalled THEN
		iDistanceMiddleDevices := REAL_TO_INT(gOverVarnish.Parameters.Hw.rOPVLength/10);
	ELSIF gDryerAnc.Parameters.xInstalled AND gOverVarnish.Parameters.xInstalled THEN
		IF gBelt.states.rCurrentSpeed > 70.0 THEN
			iDistanceMiddleDevices := REAL_TO_INT(((gDryerAnc.Parameters.Hw.rDryerLength + gOverVarnish.Parameters.Hw.rOPVLength)/10) - (2*(gBelt.states.rCurrentSpeed - 70.0)));
		ELSE
			iDistanceMiddleDevices := REAL_TO_INT((gDryerAnc.Parameters.Hw.rDryerLength + gOverVarnish.Parameters.Hw.rOPVLength)/10);
		END_IF
	END_IF

	//Define RejectDistance with distance between devices and distance in the Reject
	gThicknessCtrl.parameters.Reject.iRejectDistance := iDistanceMiddleDevices + gStacker.Parameters.Hw.iRejectAdjustmentDistance;
	gThicknessCtrl.parameters.Reject.iHoldRejectDistance := iDistanceMiddleDevices + gStacker.Parameters.Hw.iRejectAdjustmentDistance + gStacker.Parameters.Hw.iDistanceToReject;

END_ACTION

ACTION RemoteCtrl:

	IF NOT gMachine.Pt.xControlledRemotely THEN
		RETURN;
	END_IF

	tonBeltNotStopped.IN := NOT gMachine.St.Remote.xBeltNotStopped;
	tonBeltNotStopped.PT := T#1s;
	tonBeltNotStopped();

	// The signal is always TRUE, and when the belt stops, it is reseted during a second
	IF tonBeltNotStopped.Q THEN
		gMachine.St.Remote.xBeltNotStopped := TRUE;
	END_IF
	IF xBeltMovingPreviousToStop AND EDGENEG(gMachine.St.Mode.xAuto) OR EDGEPOS(gMachine.AlSummary.xAlarmStop OR gMachine.AlSummary.xAlarmCritical) THEN
		gMachine.St.Remote.xBeltNotStopped := FALSE;
	END_IF

END_ACTION
```

#### EventLog.st
```iecst
ACTION LogCriticalAlarm:

//	iReasonCritical.0 := gMachine.AlSummary.xAlrSafetySystemGeneral;
//	iReasonCritical.1 := gMachine.Al.Alarm.xAlarmSAIPowerOff;
//	iReasonCritical.2 := gBelt.AlSummary.xAlarmCritical;
//	iReasonCritical.3 := gBlock[1].AlSummary.xAlarmCritical;
//	iReasonCritical.4 := gBlock[2].AlSummary.xAlarmCritical;
//	iReasonCritical.5 := gMachine.Al.Alarm.xAlrWrongPhysConf;

	stEventLogCritical.Source := ELOG_TYPE_GENERAL;
	stEventLogCritical.Severity:= ELOG_SEVERITY_ERROR;
	stEventLogCritical.Facility:= 0;
	stEventLogCritical.ErrorCode:=0;

	stEventLogCritical.Text := 'Gen.LogCriticalAlarm';

	IF 		iReasonCritical.0 THEN stEventLogCritical.Text := 'Gen Critical. xAlrSafetySystemGeneral';
	ELSIF 	iReasonCritical.1 THEN stEventLogCritical.Text := 'Gen Critical. xAlarmSAIPowerOff';
	ELSIF 	iReasonCritical.2 THEN stEventLogCritical.Text := 'Gen Critical. Belt Crical Alarm';
	ELSIF 	iReasonCritical.3 THEN stEventLogCritical.Text := 'Gen Critical. Block 1 Critical Alarm';
	ELSIF 	iReasonCritical.4 THEN stEventLogCritical.Text := 'Gen Critical. Block 2 Critical Alarm';
	ELSIF 	iReasonCritical.5 THEN stEventLogCritical.Text := 'Gen Critical. xAlrWrongPhysConf';
	ELSIF 	iReasonCritical.6 THEN stEventLogCritical.Text := 'Gen Critical. Machine no powered';
	END_IF

	gEventLogLoader(EventData := ADR(stEventLogCritical));

END_ACTION

ACTION LogStopAlarm:

//	//Alarms stop//

//	//General 1
	stEventLog.Source := ELOG_TYPE_GENERAL;
	stEventLog.Severity:= ELOG_SEVERITY_ERROR;
	stEventLog.Facility:= 0;
	stEventLog.ErrorCode:=0;

	stEventLog.Text := 'Gen.LogStopAlarm';

	IF 		iReasonStopGen.0 THEN stEventLog.Text := 'Gen Stop. xAlarmAir1';
	ELSIF 	iReasonStopGen.1 THEN stEventLog.Text := 'Gen Stop. xAlarmComPcPLC';
	ELSIF 	iReasonStopGen.2 THEN stEventLog.Text := 'Gen Stop. xAlarmEnableWithoutBarsOn';
	ELSIF 	iReasonStopGen.3 THEN stEventLog.Text := 'Gen Stop. xAlarmMountedPiece';
	ELSIF 	iReasonStopGen.4 THEN stEventLog.Text := 'Gen Stop. xAlarmSAIPowerFault';
	ELSIF 	iReasonStopGen.5 THEN stEventLog.Text := 'Gen Stop. xAlrSafetySystemEStop';
	ELSIF 	iReasonStopGen.6 THEN stEventLog.Text := 'Gen Stop. xAlrThicknSystemNotSelected';
	ELSIF 	iReasonStopGen.7 THEN stEventLog.Text := 'Gen Stop. BK1 xAlarmStop';
	ELSIF 	iReasonStopGen.8 THEN stEventLog.Text := 'Gen Stop. BK2 xAlarmStop';
	ELSIF 	iReasonStopGen.9 THEN stEventLog.Text := 'Gen Stop. Belt xAlarmStop';
	ELSIF 	iReasonStopGen.10 THEN stEventLog.Text := 'Gen Stop. Ding xAlarmStop';
	ELSIF 	iReasonStopGen.11 THEN stEventLog.Text := 'Gen Stop. Photocell xAlarmStop';
	ELSIF 	iReasonStopGen.12 THEN stEventLog.Text := 'Gen Stop. TrVac1 xAlarmStop';
	ELSIF 	iReasonStopGen.13 THEN stEventLog.Text := 'Gen Stop. TrVac2 xAlarmStop';
	ELSIF 	iReasonStopGen.14 THEN stEventLog.Text := 'Gen Stop. xPDBrokenSensorL1';
	ELSIF 	iReasonStopGen.15 THEN stEventLog.Text := 'Gen Stop. xPDBrokenSensorL2';
	ELSIF 	iReasonStopGen.16 THEN stEventLog.Text := 'Gen Stop. Jam1 xAlarmStop';
	ELSIF 	iReasonStopGen.17 THEN stEventLog.Text := 'Gen Stop. Jam2 xAlarmStop';
	ELSIF 	iReasonStopGen.18 THEN stEventLog.Text := 'Gen Stop. NC1 xAlarmStop';
	ELSIF 	iReasonStopGen.19 THEN stEventLog.Text := 'Gen Stop. NC2 xAlarmStop';
	ELSIF 	iReasonStopGen.20 THEN stEventLog.Text := 'Gen Stop. xAlr24Vdc';
	ELSIF 	iReasonStopGen.21 THEN stEventLog.Text := 'Gen Stop. Led1 xAlarmStop';
	ELSIF 	iReasonStopGen.22 THEN stEventLog.Text := 'Gen Stop. Led2 xAlarmStop';
	ELSIF 	iReasonStopGen.23 THEN stEventLog.Text := 'Gen Stop. xAlrDingWrongPosition';
	ELSIF 	iReasonStopGen.24 THEN stEventLog.Text := 'Gen Stop. xSwCriticalCondition';
	ELSIF	iReasonStopGen.25 THEN stEventLog.Text := 'Gen Stop. Jam3 xAlarmStop';
	ELSIF	iReasonStopGen.26 THEN stEventLog.Text := 'Gen Stop. xNotLoadedImage;';
	ELSIF	iReasonStopGen.27 THEN stEventLog.Text := 'Gen Stop. CheckMedia. Possible jam';
	ELSIF	iReasonStopGen.28 THEN stEventLog.Text := 'Gen Stop. Media thickness out of limits';
	ELSIF	iReasonStopGen.29 THEN stEventLog.Text := 'Gen Stop. Media length out of limits';
	ELSIF 	iReasonStopGen.30 THEN stEventLog.Text := 'Gen Stop. Media width out of limits';
	ELSIF 	iReasonStopInks > 0 THEN stEventLog.Text := 'Gen Stop. Inks Alarm';
	END_IF

	gEventLogLoader(EventData := ADR(stEventLog));

END_ACTION

ACTION LogOutOfAuto:

//	iReasonOut.0 := gMachine.In.Buttons.xZero;
//	iReasonOut.1 := NOT gMachine.In.Buttons.xAuto AND NOT gMachine.In.Buttons.xManual; // It avoids manual state when safety is NOT ready
//	iReasonOut.2 := gMachine.AlSummary.xAlarmCritical AND (enPrinterState = PRINTERGEN_AUTO) AND NOT gMachine.St.AutoMode.xBypass;
//  iReasonOut.3 := gMachine.AlSummary.xAlrSafetySystemGeneral AND gMachine.St.Mode.xManual; //Going out of Manual just for Safety alarms

	stEventLogState.Source := ELOG_TYPE_GENERAL;
	stEventLogState.Severity:= ELOG_SEVERITY_INFO;
	stEventLogState.Facility:= 0;
	stEventLogState.ErrorCode:=0;

	stEventLogState.Text := 'Gen.OutOfMan';

	IF 		iReasonOut.0 AND gMachine.St.Mode.xManual THEN
		stEventLogState.Text := 'OutOfMan. Selector to Zero';
	ELSIF 	iReasonOut.0 AND gMachine.St.Mode.xAuto THEN
		stEventLogState.Text := 'OutOfAuto. Selector to Zero';
	ELSIF 	iReasonOut.1 AND gMachine.St.Mode.xManual THEN
		stEventLogState.Text := 'OutOfMan. Selector NOT Manual and NOT Auto';
	ELSIF 	iReasonOut.1 AND gMachine.St.Mode.xAuto THEN
		stEventLogState.Text := 'OutOfAuto. Selector NOT Manual and NOT Auto';
	ELSIF 	iReasonOut.2 THEN
		stEventLogState.Text := 'OutOfAuto. Critical Alarm';
	ELSIF 	iReasonOut.3 THEN
		stEventLogState.Text := 'OutOfMan. xAlrSafetySystemGeneral';
	END_IF

	gEventLogLoader(EventData := ADR(stEventLogState));

END_ACTION

ACTION LogAutoInProduction:

	stEventLogAutoProduction.Source := ELOG_TYPE_GENERAL;
	stEventLogAutoProduction.Severity:= ELOG_SEVERITY_INFO;
	stEventLogAutoProduction.Facility:= 0;
	stEventLogAutoProduction.ErrorCode:=0;

	stEventLogAutoProduction.Text := 'Auto in Production';

	gEventLogLoader(EventData := ADR(stEventLogAutoProduction));

END_ACTION

ACTION LogAutoInByPass:

	stEventLogAuto.Source := ELOG_TYPE_GENERAL;
	stEventLogAuto.Severity:= ELOG_SEVERITY_INFO;
	stEventLogAuto.Facility:= 0;
	stEventLogAuto.ErrorCode:=0;

	stEventLogAuto.Text := 'Auto in ByPass';

	gEventLogLoader(EventData := ADR(stEventLogAuto));

END_ACTION

ACTION LogAutoInStop:

	stEventLogAutoStop.Source := ELOG_TYPE_GENERAL;
	stEventLogAutoStop.Severity:= ELOG_SEVERITY_INFO;
	stEventLogAutoStop.Facility:= 0;
	stEventLogAutoStop.ErrorCode:=0;

	stEventLogAutoStop.Text := 'Gen.LogAutoInStop';

	IF iReasonAutoStop.0 THEN stEventLogAutoStop.Text := 'Auto in Stop: Stop signal';
	ELSIF iReasonAutoStop.1 THEN stEventLogAutoStop.Text := 'Auto in Stop: Stop by invalid automode';
	ELSIF iReasonAutoStop.2 THEN stEventLogAutoStop.Text := 'Auto in Stop: Stop without ByPass with any stop alarm';
	ELSIF iReasonAutoStop.3 THEN stEventLogAutoStop.Text := 'Auto in Stop: Stop in ByPass with thicknes sensor alarms';
	ELSIF iReasonAutoStop.4 THEN stEventLogAutoStop.Text := 'Auto in Stop: Stop in ByPass with TRansVacum stop alarm';
	ELSIF iReasonAutoStop.5 THEN stEventLogAutoStop.Text := 'Auto in Stop: Stop in ByPass with non reference vertical motor alarm';
	ELSIF iReasonAutoStop.6 THEN stEventLogAutoStop.Text := 'Auto in Stop: Stop in JamRecovery. Yimeout no action';
	ELSE stEventLogAuto.Text := 'Entgering in Auto in Stop';
	END_IF

	gEventLogLoader(EventData := ADR(stEventLogAutoStop));

END_ACTION

ACTION LogAutoInJamRecovery:

	stEventLogAutoJamRec.Source := ELOG_TYPE_GENERAL;
	stEventLogAutoJamRec.Severity:= ELOG_SEVERITY_INFO;
	stEventLogAutoJamRec.Facility:= 0;
	stEventLogAutoJamRec.ErrorCode:=0;

	stEventLogAutoJamRec.Text := 'Auto in Jam Recovery';

	gEventLogLoader(EventData := ADR(stEventLogAutoJamRec));

END_ACTION

ACTION LogAutoStart:

	stEventLogStart.Source := ELOG_TYPE_GENERAL;
	stEventLogStart.Severity:= ELOG_SEVERITY_INFO;
	stEventLogStart.Facility:= 0;
	stEventLogStart.ErrorCode:=0;

	stEventLogStart.Text := 'Auto Start Order';

	gEventLogLoader(EventData := ADR(stEventLogStart));

END_ACTION

ACTION LogAutoStop:

	stEventLogStop.Source := ELOG_TYPE_GENERAL;
	stEventLogStop.Severity:= ELOG_SEVERITY_INFO;
	stEventLogStop.Facility:= 0;
	stEventLogStop.ErrorCode:=0;

	stEventLogStop.Text := 'Auto Stop Order';

	gEventLogLoader(EventData := ADR(stEventLogStop));

END_ACTION

ACTION LogPrePrintingPos:

	stEventLogPrePrint.Source := ELOG_TYPE_GENERAL;
	stEventLogPrePrint.Severity:= ELOG_SEVERITY_INFO;
	stEventLogPrePrint.Facility:= 0;
	stEventLogPrePrint.ErrorCode:=0;

	IF iReasonForcePreprintingPos = 0 THEN
		stEventLogPrePrint.Text := 'PrePrintPos RESETED';
	ELSE
		stEventLogPrePrint.Text := 'PrePrintPos SET. Reason:';
		// Adding Reasong data to log
		brsitoa(iReasonForcePreprintingPos, ADR(strAuxEventDesc));
		brsstrcat(ADR(stEventLogPrePrint.Text), ADR(strAuxEventDesc));
	END_IF

	gEventLogLoader(EventData := ADR(stEventLogPrePrint));

END_ACTION
```

#### MachineCtrl_Fast.var - Local variables
```iecst
VAR
	xRunBeltNormal : BOOL;
	xRunBeltLab : BOOL;
	xRunBeltToBeCleaned : BOOL;
	xStopBeltWhileCleaning : BOOL;
	xSignalsStopBeltAuto : BOOL;
	xAnyTankHeaterEnabled : {REDUND_UNREPLICABLE} BOOL;
	xUserRaisesBlocks : BOOL;
	xOrdersRunBeltNormal : BOOL;
	xRunBeltByPass : BOOL;
	xInCap : BOOL;
	xGoingToCap : BOOL;
	xGoingToPrint : BOOL;
	xCleaning : BOOL;
	xInPrint : BOOL;
	xAlarmToEmpyBelt : BOOL;
	xAlarmsStopBeltRun : BOOL;
	enPrinterState : enumEFI_GenMachineState := PRINTERGEN_ZERO; (*PRINTERGEN_ZERO*)
	enPrinterStatesInAuto : enumEFI_MachineState := PRINTERGEN_ZERO; (*PRINTERGEN_ZERO*)
	rsRunBeltOrderManual : RS;
	srStopBeltNoImage : SR;
	srPauseMachine : {REDUND_UNREPLICABLE} RS;
	stPrinterAlarmsSummaryReseted : stEFI_AlarmSummary; (*stDingAlarmsReseted : stPhotoCellsAlarms;*)
	stPrinterAlarmsReseted : StGeneral_Alarms;
	stPrinterAlarmsListReseted : StGeneral_AlarmsList;
	tofMachineCleaning : TOF;
	tonStartButton : TON;
	ton_ZeroMode : TON;
	ton_JamRecoveryIdle : TON;
	T_AlarmPDL2 : TON;
	T_AlarmPDL1 : TON;
	TP_AlrBentTile : TP;
	iIndexReviewArray : UINT;
	iIndexCuringBar : USINT;
	iIndexBlock : USINT;
	iReasonOut : UDINT;
	iReasonStopInks : UDINT;
	iReasonStopGen : UDINT;
	iReasonCritical : UDINT;
	stEventLogAutoJamRec : EventLog_typ;
	stEventLogAutoProduction : EventLog_typ;
	stEventLogAutoStop : EventLog_typ;
	stEventLogAuto : EventLog_typ;
	stEventLogState : EventLog_typ;
	stEventLogCritical : EventLog_typ;
	stEventLog : EventLog_typ;
	stEventLogStart : EventLog_typ;
	stEventLogStop : EventLog_typ;
	stEventLogPrePrint : EventLog_typ;
	g_xRunBeltOrderManual : BOOL; (*Belt order in manual filtered*)
	g_xRunBeltOrderAuto : BOOL; (*Belt order in auto*)
	reasonAnyWarningInks : UINT;
	reasonAnyWarningGen : UDINT;
	tonResetCmd : TON;
	xEnabledAlarmPDSensor1 : BOOL;
	xEnabledAlarmPDSensor2 : BOOL;
	usiIndex : USINT;
	xForcePreprintingPos : BOOL;
	iReasonForcePreprintingPos : USINT;
	iPrevReasonForcePreprintingPos : USINT;
	iReasonStopBeltAuto : USINT;
	InputsSwReseted : stGeneral_Inputs_Sw;
	tonDelayToSafetyPos : TON;
	srUpBarsToSafePos : SR;
	xMachReadyToPrint : BOOL; (*In print postion without safe offsets position*)
	xRunBeltByLine : BOOL;
	iReasonAutoStop : UINT;
	iReasonAutoStop_Trigger : UINT;
	iReasonAutoCmdStart : UINT;
	iReasonAutoCmdStop : UINT;
	iReasonAutoCmdStop_Trigger : UINT;
	xOrderToCapReceived : BOOL;
	xOrderToPrintReceived : BOOL;
	iReasonCap : UINT;
	iReasonPrint : UINT;
	lastReasonCap : UINT;
	iBlockExecutionsOrder : UDINT;
	lastReasonPrint : UINT;
	iBlockDelay : UDINT;
	iReasonSetPause : UINT;
	iReasonResetPause : UINT;
	iLastReasonSetPause : UINT;
	iLastReasonResetPause : UINT;
	TOF_AlarmDingPosition : TOF;
	iReasonSafetySystemGeneral : UINT;
	iReasonSafetyCutAir : UINT;
	tonResetCommandIcla : TON;
	xStopBeltJamTesting : BOOL; (*Jam detect system is in testing proces, wait finish to start belt*)
	xPrintShootingForced : BOOL; (*Print shoot by instantprint or continousprint active*)
	xMediaThicknessModified : BOOL;
	rPrevMediaThickness : REAL;
	xMachineRaisesBlock : BOOL;
	BoardsFeedMinGap : BlinkOnOff;
	tiBoardTime : TIME;
	tiGapTime : TIME;
	rBeltSpeedMmMs : REAL; (*Belt speed in mm/ms*)
	rPrevBoardLength : REAL;
	rPrevBoardGap : REAL;
	rPrevStainLength : REAL;
	rPrevStainGap : REAL;
	rPrevBeltSpeed : REAL;
	xFormatChanged : BOOL;
	xBeltSpeedChanged : BOOL;
	tofToAutoAfterEnableSafety : TOF;
	tofResetAfterEnableSafety : TOF;
	tofResetFromUI : TOF;
	TON_AlrDegasserPressure : TON;
	iReasonRunBlowerRemote : USINT;
	iReasonOrdersRunBeltProduction : USINT;
	iReasonORunBeltPhoto : BOOL;
	iDistanceMiddleDevices : INT;
	xSensorIncoherenceDetectedL1 : BOOL;
	xSensorIncoherenceDetectedL2 : BOOL;
	diCountProductDetectEdgesL1 : UDINT;
	diCountProductDetectEdgesL2 : UDINT;
	xUseBelowSensorToApplyOffset : BOOL;
	xUseAboveSensorToApplyOffset : BOOL;
	xMediaInLedPosition : BOOL;
	iReasonRunNitrogenFlow : USINT;
	xPDSignalSensorL1 : REFERENCE TO BOOL; (*Use just in MachineInputs*)
	xPDSignalSensorL2 : REFERENCE TO BOOL; (*Use just in MachineInputs*)
	xPDCarriageL1 : REFERENCE TO BOOL; (*Use just in MachineInputs*)
	xPDCarriageL2 : REFERENCE TO BOOL; (*Use just in MachineInputs*)
	tonRaiseBarsInPause : TON;
	tonProtecPHBlowers : TON;
	xReasonRunVacuumProduction : USINT;
	tonResetSendingJob : TON;
	xStartVacuumWhileGoingDown : BOOL;
	tonEnterSafety : TON;
	xEdgeSafety : BOOL;
	xCuringDesired : ARRAY[0..MAX_LAST_CURING_LED] OF BOOL;
	tonBeltNotStopped : TON;
	xBeltMovingPreviousToStop : BOOL;
	strAuxEventDesc : STRING[129];
	rMountedLimit : REAL;
	rCoef : REAL; (*Coeficient to be applied to setpoint from SW*)
END_VAR
```

### Program Logical/Printer/MachineCtrl/MachineCtrl_Slow (IEC)
